Yaskawa INFORM job: SKRZYNIA_5440_180_STOPNI_10B_NEW.JBI

/JOB
//NAME SKRZYNIA_5440_180_STOPNI_10B_NEW
///FOLDERNAME 02-SKRZYNIE_JOBS
//POS
///NPOS 748,748,0,32,0,0
///TOOL 0
///POSTYPE PULSE
///PULSE
C00000=-21231,-51303,42314,2367,6591,-1439
C00001=-12854,-61498,-6635,149088,-29435,16513
C00002=84284,-61498,-6635,149088,14842,16513
C00003=84426,-61498,-62039,149088,14842,16513
C00004=84426,-61498,-83719,149088,14842,16513
C00005=40079,-25830,-61904,72398,37828,17494
C00006=40079,-25830,-61904,72398,37828,17494
C00007=38824,-23395,-60038,72349,38727,17731
C00008=41545,-22667,-59464,70826,37145,18191
C00009=40079,-25830,-61904,72398,37828,17494
C00010=40079,-23879,-31232,97616,36989,2612
C00011=40241,-22903,-30855,97033,36795,2952
C00012=39596,-21803,-29985,96678,37187,3182
C00013=41542,-21522,-29763,96797,35874,3054
C00014=40241,-22903,-30855,97033,36795,2952
C00015=44500,-22967,-34027,49689,40772,15208
C00016=44759,-21950,-33222,49364,40770,15399
C00017=43898,-20603,-32137,49608,41392,15289
C00018=45676,-20288,-31878,48567,40497,15854
C00019=44759,-21950,-33222,49364,40770,15399
C00020=50639,-31838,-53853,40430,42590,20636
C00021=47737,-42531,-47731,84740,46626,-3202
C00022=73324,-51450,-15857,136644,48513,-27329
C00023=28578,-31257,-33285,101874,54895,-3139
C00024=29101,-23166,-41439,93785,52323,3372
C00025=30342,-16402,-40775,90158,51109,6027
C00026=29555,-14242,-38855,90054,51607,6222
C00027=31304,-14182,-38798,89754,50458,6198
C00028=30342,-16402,-40775,90158,51109,6027
C00029=37840,-26567,-47806,97824,39338,5403
C00030=38314,-22656,-45541,96192,38787,6352
C00031=38740,-21749,-44817,95954,38481,6451
C00032=38106,-20505,-43805,95701,38856,6673
C00033=39920,-20274,-43616,95549,37666,6573
C00034=38740,-21749,-44817,95954,38481,6451
C00035=35154,-23288,-28184,89821,43405,2441
C00036=35403,-21021,-26397,89340,43215,2751
C00037=34678,-19569,-25213,89063,43699,2948
C00038=36545,-19419,-25091,89018,42427,2940
C00039=35403,-21021,-26397,89340,43215,2751
C00040=46673,-28267,-59493,36306,49500,22578
C00041=47298,-25083,-54483,36432,48421,22382
C00042=46134,-23276,-53085,36983,49197,22170
C00043=48093,-22778,-52692,35651,48513,22818
C00044=47298,-25083,-54483,36432,48421,22382
C00045=43000,-32780,-49011,53703,41088,15214
C00046=66148,-65994,-55487,105361,28212,-7739
C00047=66148,-65994,-55487,105361,28212,-7739
C00048=59848,-54778,-49507,133915,29212,-10807
C00049=45497,-38347,-41839,114412,32622,-465
C00050=46376,-32635,-46933,102993,29107,5780
C00051=46303,-28031,-46898,97061,28371,8976
C00052=45038,-26161,-45521,96183,29128,9541
C00053=46946,-25787,-45238,96120,27855,9431
C00054=46303,-28031,-46898,97061,28371,8976
C00055=45864,-17128,1685,129467,40696,-9274
C00056=46023,-15894,1830,128891,40053,-8896
C00057=45181,-14790,2774,128176,40341,-8535
C00058=46921,-14545,2986,129317,39465,-9073
C00059=45402,-17127,796,128656,40504,-8810
C00060=42828,-21985,-11573,106778,34538,-1929
C00061=43349,-21404,-11124,106831,34165,-1930
C00062=42250,-19876,-9917,105946,34757,-1485
C00063=44494,-19460,-9583,106781,33302,-1837
C00064=42797,-21858,-11474,106726,34550,-1903
C00065=42956,-14057,7354,88292,32197,-569
C00066=43438,-13569,7781,88275,31880,-510
C00067=42549,-12302,8904,87823,32462,-349
C00068=44721,-11883,9282,88161,31033,-316
C00069=42944,-14884,6642,88491,32210,-682
C00070=72417,-64226,-72669,53660,37323,27470
C00071=81480,-74508,-67932,111005,17511,3722
C00072=42492,-36415,-29790,92406,42740,11684
C00073=29699,-14901,-14062,86637,51249,15251
C00074=28921,-12904,-12269,86425,51786,15406
C00075=30978,-12767,-12144,86426,50380,15429
C00076=29506,-17416,-16239,86937,51377,15018
C00077=29506,-17416,-16239,86937,51377,15018
C00078=44296,-22319,-14791,77397,31382,16857
C00079=44081,-20100,-12685,77077,31564,17025
C00080=42936,-18463,-11353,76734,32387,17168
C00081=44621,-18276,-11197,76464,31271,17386
C00082=44081,-20100,-12685,77077,31564,17025
C00083=88410,-69609,-60867,139529,19008,-8209
C00084=82254,-59190,-37505,135829,26015,-2584
C00085=48709,-26647,-10027,118963,31871,904
C00086=44740,-24992,-19428,105622,30913,8023
C00087=35836,-10089,175,120717,54219,3716
C00088=33571,-11609,-5533,116057,52820,8482
C00089=32638,-9483,-3533,115639,53262,8773
C00090=34483,-9329,-3384,116184,52162,8425
C00091=33571,-11609,-5533,116057,52820,8482
C00092=29299,-14235,-8112,85858,51306,13749
C00093=30258,-13056,-7056,85778,50658,13854
C00094=29454,-11053,-5212,85557,51212,13988
C00095=31306,-10982,-5149,85624,49953,14016
C00096=30258,-13056,-7056,85778,50658,13854
C00097=44150,-27478,-14760,79983,38437,11062
C00098=60260,-41997,-20174,82745,25327,6782
C00099=62412,-62489,-12046,-12266,17816,34850
C00100=0,-52280,40443,0,6876,0
C00101=-681,-52632,38645,-5695,5489,-631
C00102=-17840,-61498,-6635,-149088,-29435,-16513
C00103=-84284,-61498,-6635,-149088,14842,-16513
C00104=-84426,-61498,-62039,-149088,14842,-16513
C00105=-84426,-61498,-83719,-149088,14842,-16513
C00106=-83351,-27062,-60322,-167360,37385,6517
C00107=-83351,-27062,-60322,-167360,37385,23281
C00108=-45097,-23850,-79932,-76262,26943,-22849
C00109=-48253,-15729,-73342,-71138,25693,-24842
C00110=-50302,-13076,-73239,-65836,25323,-27140
C00111=-49401,-11675,-71961,-66260,25816,-27133
C00112=-50608,-11574,-71867,-65226,25249,-27391
C00113=-49660,-13361,-73494,-66442,25615,-26975
C00114=-48242,-21102,-77802,-73044,25430,-23851
C00115=-42432,-29691,-46140,-101591,34194,-3953
C00116=-40467,-32259,-45349,-89481,35752,-6083
C00117=-35590,-22323,-38089,-87474,43148,-7978
C00118=-34853,-20780,-36847,-87247,43643,-8181
C00119=-37029,-20471,-36594,-86926,42180,-8224
C00120=-35503,-23333,-38886,-87700,43207,-7835
C00121=-41659,-25848,-37197,-61468,39541,-12344
C00122=-42019,-23363,-32043,-63110,38591,-11327
C00123=-41283,-22167,-31102,-63128,39154,-11341
C00124=-43189,-21868,-30866,-62281,38009,-11788
C00125=-40846,-25460,-35158,-62968,39555,-11455
C00126=-39561,-32409,-42051,-71473,38885,-9254
C00127=-88477,-67032,-53890,-125185,13082,17955
C00128=-90715,-66667,-50935,-152816,24533,28486
C00129=-30735,-26920,-32844,-95116,50209,-1071
C00130=-37180,-24683,-31930,-114741,47007,2943
C00131=-36407,-19634,-34656,-109847,45004,-453
C00132=-38352,-16604,-33863,-108521,43129,-1176
C00133=-37479,-14809,-32279,-108169,43576,-1482
C00134=-39395,-14487,-31992,-108361,42368,-1194
C00135=-37253,-18321,-35339,-108644,43916,-1187
C00136=-30948,-19486,-27368,-89515,49970,-2899
C00137=-32453,-17458,-25663,-89179,48933,-3088
C00138=-31896,-16151,-24534,-89028,49305,-3221
C00139=-33527,-16125,-24510,-88960,48196,-3202
C00140=-31291,-18911,-26892,-89421,49733,-2955
C00141=-32789,-14788,-10714,-75998,48642,-1904
C00142=-33953,-13481,-9550,-75758,47902,-2112
C00143=-33380,-12226,-8408,-75670,48319,-2157
C00144=-35020,-12164,-8351,-75529,47228,-2306
C00145=-33300,-14767,-10697,-75957,48300,-1949
C00146=-33300,-14767,-10697,-75957,48300,-1949
C00147=-33901,-13199,-7224,-76945,47663,-1266
C00148=-33178,-11617,-5779,-76815,48184,-1329
C00149=-35129,-11426,-5603,-76688,46886,-1497
C00150=-32900,-14718,-9841,-76444,48459,-1584
C00151=-46324,-38325,-53351,-48650,39022,-16558
C00152=-84678,-53272,-42524,-56273,5220,-14251
C00153=-79949,-57830,-54545,-43165,18800,-25262
C00154=-85199,-63426,-59279,-35356,8253,-25340
C00155=-43240,-40066,-69296,-76804,34492,-13950
C00156=-32352,-24302,-62495,-76398,48702,-17646
C00157=-33867,-19497,-59989,-74208,48202,-18898
C00158=-33043,-17469,-58279,-74274,48770,-19034
C00159=-35172,-17180,-58031,-73305,47532,-19251
C00160=-33150,-20833,-61090,-74721,48572,-18687
C00161=-32525,-19963,-22291,-97454,48417,-2656
C00162=-34479,-17146,-19937,-97221,47013,-2812
C00163=-33716,-15515,-18525,-96928,47480,-3025
C00164=-35357,-15455,-18472,-97073,46375,-2908
C00165=-33341,-18474,-21063,-97306,47817,-2759
C00166=-32838,-10388,7981,-94473,48357,2926
C00167=-33747,-9461,8037,-94117,47673,2571
C00168=-33094,-8062,9377,-93861,48090,2458
C00169=-34952,-7927,9507,-94260,46861,2543
C00170=-33010,-10379,7174,-94037,48174,2591
C00171=-36099,-20774,-22249,-70758,44565,-7624
C00172=-37926,-16067,-12890,-73276,42575,-5996
C00173=-37323,-14944,-11908,-73188,43017,-6038
C00174=-39053,-14785,-11769,-72915,41882,-6255
C00175=-37847,-19214,-17221,-72670,42783,-6386
C00176=-73757,-59015,-49060,-81128,17325,-3444
C00177=-66351,-49775,-22313,-134939,32824,19491
C00178=-38126,-18978,-6321,-103556,42156,4232
C00179=-39485,-17529,-8330,-90200,39091,223
C00180=-38315,-15563,-6658,-89669,39866,-39
C00181=-40130,-15376,-6497,-89855,38637,-21
C00182=-40610,-23081,-12745,-91737,38407,1092
C00183=-40833,-20771,-16117,-71062,38118,-5732
C00184=-41179,-17944,-14058,-70159,38104,-6286
C00185=-40208,-16344,-12701,-70049,38815,-6328
C00186=-42019,-16101,-12492,-69614,37653,-6637
C00187=-41179,-17944,-14058,-70159,38104,-6286
C00188=-82794,-45547,-18103,-153793,26453,27163
C00189=-59391,-59726,-723,-139936,47315,26256
C00190=-59391,-63256,-7305,-138930,45803,25558
C00191=-41911,-25348,-18707,-96909,37821,5942
C00192=-39278,-18921,-13723,-94727,39374,4724
C00193=-50267,-3803,20766,-145166,53580,20077
C00194=-49199,-2294,22340,-144514,53890,19722
C00195=-50839,-1881,22778,-145489,53339,20243
C00196=-50267,-457,30009,-146420,56926,21139
C00197=-39278,-18921,-13723,-94727,39374,4724
C00198=-38355,-17353,-12416,-94258,39960,4466
C00199=-40180,-17161,-12255,-94505,38724,4557
C00200=-37963,-22229,-16363,-95272,40353,5112
C00201=-56568,-73357,-35482,-123268,35826,13545
C00202=-46099,-67236,-11725,-98004,28606,19827
C00203=275,-40498,62911,330,272,-175
C00204=-21231,-51303,42314,2367,6591,-1439
C00205=-12854,-61498,-6635,149088,-29435,16513
C00206=84284,-61498,-6635,149088,14842,16513
C00207=84426,-61498,-62039,149088,14842,16513
C00208=84426,-61498,-83719,149088,14842,16513
C00209=40079,-25830,-61904,72398,37828,17494
C00210=43542,-21744,-53414,85694,32141,12908
C00211=43538,-20959,-59091,78847,32551,16732
C00212=40079,-23879,-31232,97616,36989,2612
C00213=41069,-22296,-36683,87871,35939,7163
C00214=41069,-20857,-27994,94343,36275,3375
C00215=40241,-22903,-30855,97033,36795,2952
C00216=44500,-22967,-34027,49689,40772,15208
C00217=37674,-14410,-29425,54908,51799,12689
C00218=37617,-13106,-20810,58248,49229,10178
C00219=44759,-21950,-33222,49364,40770,15399
C00220=50639,-31838,-53853,40430,42590,20636
C00221=47737,-42531,-47731,84740,46626,-3202
C00222=78713,-49095,-28754,133607,38203,-24422
C00223=28578,-31257,-33285,101874,54895,-3139
C00224=29101,-23166,-41439,93785,52323,3372
C00225=31163,-13872,-34138,92103,50752,4440
C00226=31163,-14064,-41434,88282,50498,7326
C00227=30342,-16402,-40775,90158,51109,6027
C00228=37840,-26567,-47806,97824,39338,5403
C00229=38314,-22656,-45541,96192,38787,6352
C00230=39658,-19881,-39017,99036,38353,4498
C00231=39658,-20227,-46296,93241,37598,7980
C00232=38740,-21749,-44817,95954,38481,6451
C00233=35154,-23288,-28184,89821,43405,2441
C00234=36302,-20456,-32356,81251,42995,6506
C00235=36302,-19046,-24537,85721,42698,3608
C00236=35403,-21021,-26397,89340,43215,2751
C00237=46673,-28267,-59493,36306,49500,22578
C00238=35383,-14910,-45807,52457,59655,19882
C00239=35383,-15025,-38926,54776,56903,17744
C00240=47298,-25083,-54483,36432,48421,22382
C00241=43000,-32780,-49011,53703,41088,15214
C00242=90538,-65158,-52413,145953,6697,-22013
C00243=90538,-65158,-52413,145953,6697,-22013
C00244=59848,-54778,-49507,133915,29212,-10807
C00245=45497,-38347,-41839,114412,32622,-465
C00246=46376,-32635,-46933,102993,29107,5780
C00247=38443,-20223,-37840,96971,39567,10287
C00248=38443,-20698,-44956,91660,38993,13539
C00249=46303,-28031,-46898,97061,28371,8976
C00250=45864,-17128,1685,129467,40696,-9274
C00251=38069,-7942,12691,120284,49952,-5070
C00252=38069,-11604,1369,116685,47266,-2469
C00253=45402,-17127,796,128656,40504,-8810
C00254=42828,-21985,-11573,106778,34538,-1929
C00255=33281,-15275,-13406,92642,47209,4970
C00256=33281,-12456,-2996,97026,47894,1870
C00257=42797,-21858,-11474,106726,34550,-1903
C00258=42956,-14057,7354,88292,32197,-569
C00259=35915,-8349,8335,81338,43542,2014
C00260=35915,-4149,20758,86814,43229,-1568
C00261=42944,-14884,6642,88491,32210,-682
C00262=72417,-64226,-72669,53660,37323,27470
C00263=81480,-74508,-67932,111005,17511,3722
C00264=42492,-36415,-29790,92406,42740,11684
C00265=30589,-12517,-11440,90322,50747,14596
C00266=30928,-12247,-10742,85035,50377,15419
C00267=29506,-17416,-16239,86937,51377,15018
C00268=33836,-18112,-25401,68178,50408,21159
C00269=33465,-13162,-18426,69063,50292,20506
C00270=33465,-11483,-10771,72168,49104,18208
C00271=88410,-69609,-60867,139529,19008,-8209
C00272=82254,-59190,-37505,135829,26015,-2584
C00273=48709,-26647,-10027,118963,31871,904
C00274=44740,-24992,-19428,105622,30913,8023
C00275=35836,-10089,175,120717,54219,3716
C00276=34345,-8030,793,117331,53206,7509
C00277=34322,-10419,-8163,114502,51063,9720
C00278=33571,-11609,-5533,116057,52820,8482
C00279=29299,-14235,-8112,85858,51306,13749
C00280=31207,-11656,-8788,84025,50108,15207
C00281=31207,-8775,1760,88103,49995,12167
C00282=30258,-13056,-7056,85778,50658,13854
C00283=44150,-27478,-14760,79983,38437,11062
C00284=60260,-41997,-20174,82745,25327,6782
C00285=62412,-62489,-12046,-12266,17816,34850
C00286=0,-52280,40443,0,6876,0
C00287=-681,-52632,38645,-5695,5489,-631
C00288=-17840,-61498,-6635,-149088,-29435,-16513
C00289=-84284,-61498,-6635,-149088,14842,-16513
C00290=-84426,-61498,-62039,-149088,14842,-16513
C00291=-84426,-61498,-83719,-149088,14842,-16513
C00292=-83351,-27062,-60322,-167360,37385,6517
C00293=-83351,-27062,-60322,-167360,37385,23281
C00294=-45097,-23850,-79932,-76262,26943,-22849
C00295=-48253,-15729,-73342,-71138,25693,-24842
C00296=-42869,-6204,-67496,-75794,33821,-25861
C00297=-42869,-3205,-70686,-69723,34977,-29338
C00298=-49660,-13361,-73494,-66442,25615,-26975
C00299=-48242,-21102,-77802,-73044,25430,-23851
C00300=-42432,-29691,-46140,-101591,34194,-3953
C00301=-40467,-32259,-45349,-89481,35752,-6083
C00302=-32032,-15700,-34761,-86363,49905,-9645
C00303=-32032,-14866,-27372,-89947,49973,-6979
C00304=-35503,-23333,-38886,-87700,43207,-7835
C00305=-41659,-25848,-37197,-61468,39541,-12344
C00306=-32550,-13183,-23016,-68651,53358,-8526
C00307=-34023,-12481,-22084,-63241,53452,-9524
C00308=-40846,-25460,-35158,-62968,39555,-11455
C00309=-39561,-32409,-42051,-71473,38885,-9254
C00310=-88477,-67032,-53890,-125185,13082,17955
C00311=-90715,-66667,-50935,-152816,24533,28486
C00312=-30735,-26920,-32844,-95116,50209,-1071
C00313=-37180,-24683,-31930,-114741,47007,2943
C00314=-36407,-19634,-34656,-109847,45004,-453
C00315=-39264,-14095,-28560,-110319,43249,69
C00316=-39254,-14742,-35710,-105973,41627,-2729
C00317=-37253,-18321,-35339,-108644,43916,-1187
C00318=-30948,-19486,-27368,-89515,49970,-2899
C00319=-33188,-17217,-33290,-80523,49125,-7157
C00320=-33231,-16133,-25752,-84153,48705,-4513
C00321=-31291,-18911,-26892,-89421,49733,-2955
C00322=-32789,-14788,-10714,-75998,48642,-1904
C00323=-32456,-10000,-8763,-74569,51725,-2878
C00324=-32456,-7502,814,-78111,50801,-165
C00325=-33300,-14767,-10697,-75957,48300,-1949
C00326=-33300,-14767,-10697,-75957,48300,-1949
C00327=-31039,-7597,-4415,-75714,54029,-1891
C00328=-31745,-5891,1281,-74609,53027,-1007
C00329=-32900,-14718,-9841,-76444,48459,-1584
C00330=-46324,-38325,-53351,-48650,39022,-16558
C00331=-84678,-53272,-42524,-56273,5220,-14251
C00332=-79949,-57830,-54545,-43165,18800,-25262
C00333=-85199,-63426,-59279,-35356,8253,-25340
C00334=-43240,-40066,-69296,-76804,34492,-13950
C00335=-32352,-24302,-62495,-76398,48702,-17646
C00336=-34311,-15084,-43386,-89458,46770,-12174
C00337=-34303,-14562,-49859,-85086,46777,-15220
C00338=-33150,-20833,-61090,-74721,48572,-18687
C00339=-32525,-19963,-22291,-97454,48417,-2656
C00340=-35706,-13608,-12356,-102024,46946,-662
C00341=-35706,-15621,-21438,-97808,45877,-3577
C00342=-33341,-18474,-21063,-97306,47817,-2759
C00343=-32838,-10388,7981,-94473,48357,2926
C00344=-33093,-7396,5806,-90907,49596,566
C00345=-33114,-3922,16616,-94789,50065,3444
C00346=-33010,-10379,7174,-94037,48174,2591
C00347=-36099,-20774,-22249,-70758,44565,-7624
C00348=-34715,-11750,-12273,-72011,49148,-6727
C00349=-34715,-9605,-3694,-75523,48112,-4187
C00350=-37847,-19214,-17221,-72670,42783,-6386
C00351=-73757,-59015,-49060,-81128,17325,-3444
C00352=-66351,-49775,-22313,-134939,32824,19491
C00353=-38126,-18978,-6321,-103556,42156,4232
C00354=-35411,-10902,-672,-92816,45935,848
C00355=-36000,-11295,-2683,-84848,44809,-1301
C00356=-40610,-23081,-12745,-91737,38407,1092
C00357=-46116,-25645,-29995,-54013,38610,-12898
C00358=-36364,-11468,-16502,-61524,50356,-10311
C00359=-36364,-9268,-6699,-65335,48232,-7516
C00360=-35369,-17970,-15673,-74843,50412,-3942
C00361=-82794,-45547,-18103,-153793,26453,27163
C00362=-59391,-59726,-723,-139936,47315,26256
///LIMIT ON
C00363=-59391,-69594,-18878,-137021,43274,24283
///LIMIT OFF
C00364=-41911,-25348,-18707,-96909,37821,5942
C00365=-39278,-18921,-13723,-94727,39374,4724
C00366=-41964,3488,28151,-134521,60914,14195
C00367=-41964,-819,15200,-132329,56719,12142
C00368=-50267,-457,30009,-146420,56926,21139
C00369=-33715,-10212,-1364,-94538,48612,5206
C00370=-33715,-12585,-10220,-90890,48191,2581
C00371=-37963,-22229,-16363,-95272,40353,5112
C00372=-66368,-73811,-34662,-141094,38161,28545
C00373=-46099,-67236,-11725,-98004,28606,19827
C00374=275,-40498,62911,330,272,-175
C00375=-21231,-51303,42314,2367,6591,-1439
C00376=-12854,-61498,-6635,149088,-29435,16513
C00377=32880,-72586,-50560,79734,53940,25582
C00378=76664,-93599,-96338,114349,24908,7990
C00379=72545,-76403,-90681,98079,12187,16258
C00380=68435,-42241,-79282,43384,21203,43145
C00381=65057,-16377,-54230,51764,24572,24912
C00382=65057,-16377,-54230,51764,24572,24912
C00383=63338,-14509,-52578,53100,25585,24479
C00384=65493,-13068,-51269,50530,24633,25485
C00385=65057,-16377,-54230,51764,24572,24912
C00386=65057,-15356,-24189,99795,20011,765
C00387=64877,-14372,-23690,98704,20045,1316
C00388=64002,-13489,-22890,98156,20604,1621
C00389=65592,-12702,-22173,98357,19527,1466
C00390=64877,-14372,-23690,98704,20045,1316
C00391=68341,-13254,-25781,29903,31229,25524
C00392=68283,-12212,-24821,29865,31356,25548
C00393=67188,-11145,-23825,30867,31841,25051
C00394=68624,-10377,-23095,29361,31405,25809
C00395=68283,-12212,-24821,29865,31356,25548
C00396=67373,-28813,-51747,26561,36937,27500
C00397=65665,-56911,-59086,75825,31170,1181
C00398=86238,-56758,-47218,93606,16664,-7096
C00399=86238,-56758,-47218,93606,16664,-7096
C00400=58162,-25487,-29222,106212,35121,-6052
C00401=54729,-17550,-36821,90686,35172,3055
C00402=53879,-10723,-35593,84994,35691,6442
C00403=52628,-8898,-33837,85063,36512,6546
C00404=54193,-8333,-33282,84633,35489,6620
C00405=53879,-10723,-35593,84994,35691,6442
C00406=63265,-18185,-41125,95483,22448,4389
C00407=62561,-14368,-38517,92984,22773,5727
C00408=62689,-13396,-37636,92694,22678,5861
C00409=61812,-12400,-36718,92465,23238,6064
C00410=63331,-11679,-36046,92201,22238,6052
C00411=62689,-13396,-37636,92694,22678,5861
C00412=60836,-16142,-22303,87853,25853,3109
C00413=60346,-13901,-20318,87240,26185,3441
C00414=59279,-12702,-19226,86999,26911,3593
C00415=60868,-12050,-18626,86765,25831,3679
C00416=60346,-13901,-20318,87240,26185,3441
C00417=71174,-16943,-50501,16787,44328,31924
C00418=70846,-13961,-45205,17496,43056,31510
C00419=69412,-12602,-43961,18675,43507,30969
C00420=70949,-11616,-43043,17320,43301,31610
C00421=70846,-13961,-45205,17496,43056,31510
C00422=66765,-25643,-43957,33958,30926,25005
C00423=89904,-51519,-74342,14421,36812,44678
C00424=59533,-60921,-66479,83565,41795,11392
C00425=74572,-27669,-34920,136415,14797,-11887
C00426=72479,-21736,-38943,108586,11547,1590
C00427=70901,-17325,-38411,94105,11830,8638
C00428=69318,-15905,-37172,92885,12849,9347
C00429=70820,-15051,-36412,92531,11846,9399
C00430=70901,-17325,-38411,94105,11830,8638
C00431=70927,-7523,10343,151197,29871,-19432
C00432=70517,-6236,10737,150221,29352,-18933
C00433=69462,-5331,11645,148944,29606,-18324
C00434=70849,-4645,12343,150548,29173,-19084
C00435=70402,-7634,9356,150158,29478,-18907
C00436=68660,-13051,-4106,122816,18275,-8999
C00437=68895,-12351,-3471,122899,18094,-9031
C00438=67458,-11121,-2337,120787,18802,-8043
C00439=69212,-10147,-1425,122703,17774,-8922
C00440=68590,-12934,-4000,122687,18305,-8939
C00441=67960,-5141,15741,92957,15720,-628
C00442=68207,-4523,16370,92944,15555,-601
C00443=67051,-3465,17460,92338,16311,-404
C00444=68762,-2475,18496,92897,15183,-531
C00445=68227,-5981,14898,93242,15553,-745
C00446=75423,-38775,-29488,68062,11357,11878
C00447=83800,-53438,-37305,103753,14733,-1265
C00448=73693,-37430,-30368,101200,21937,8332
C00449=54083,-9583,-9164,86048,34613,15862
C00450=52816,-7862,-7494,85864,35484,15962
C00451=54627,-7152,-6792,85763,34247,16030
C00452=54668,-12069,-11504,86415,34208,15656
C00453=56304,-11796,-18615,61131,36292,25169
C00454=55378,-9761,-17250,60867,37124,25353
C00455=54231,-8210,-15746,61227,37881,25175
C00456=56022,-7436,-14984,60355,36824,25634
C00457=55378,-9761,-17250,60867,37124,25353
C00458=89016,-59505,-36896,143842,20811,-11822
C00459=60495,-76741,-47652,120298,37447,-3273
C00460=76037,-16315,-2108,148598,17507,-12246
C00461=70560,-15452,-11753,122116,14270,428
C00462=55952,-2531,9844,130476,44298,-1945
C00463=56211,-3395,4409,126223,41962,1193
C00464=55729,-3443,2508,124592,39934,3479
C00465=57337,-2775,3210,125461,39069,2998
C00466=55715,-2364,6430,126525,43399,286
C00467=54062,-9026,-3291,86300,34474,14396
C00468=54568,-7612,-1915,86151,34132,14497
C00469=53276,-5879,-187,85948,35014,14576
C00470=54919,-5291,406,85945,33897,14626
C00471=54568,-7612,-1915,86151,34132,14497
C00472=55516,-30048,-16468,81245,30784,11190
C00473=78642,-41617,-20006,83725,13431,8209
C00474=0,-52280,40443,0,6876,0
C00475=-681,-52632,38645,-5695,5489,-631
C00476=-17840,-61498,-6635,-149088,-29435,-16513
C00477=-84284,-61498,-6635,-149088,14842,-16513
C00478=-57949,-92832,-68327,-119114,39180,-13331
C00479=-51160,-78996,-68705,-103851,38676,-21739
C00480=-70129,-12201,-70194,-45988,15849,-32683
C00481=-70861,-4247,-62448,-43170,16032,-33903
C00482=-72229,-1292,-61598,-37253,16795,-36501
C00483=-71164,-286,-60510,-39045,17142,-35862
C00484=-72168,114,-60071,-37345,16819,-36474
C00485=-71747,-1710,-62044,-38091,16943,-36199
C00486=-72086,-8949,-67137,-41785,15362,-34318
C00487=-68226,-19972,-38714,-103620,16923,-1218
C00488=-67549,-22986,-38612,-80975,17520,-9124
C00489=-60286,-14955,-31870,-81576,26630,-9634
C00490=-59206,-13694,-30736,-81541,27366,-9725
C00491=-61026,-12796,-29913,-80837,26167,-9971
C00492=-60502,-15936,-32740,-81790,26471,-9505
C00493=-66711,-16726,-29834,-42060,26790,-21996
C00494=-66477,-14329,-24475,-44917,25565,-20507
C00495=-65503,-13376,-23611,-45716,26132,-20127
C00496=-67048,-12587,-22889,-44009,25442,-20959
C00497=-66009,-16611,-27996,-44380,26285,-20808
C00498=-67084,-23473,-35621,-52822,22843,-18344
C00499=-54372,-63877,-56403,-90862,27079,1323
C00500=-55608,-75012,-34654,-126966,55573,20814
C00501=-55608,-75012,-34654,-126966,55573,20814
C00502=-58069,-20780,-28125,-95622,31565,-134
C00503=-62818,-16895,-25617,-123146,31403,8811
C00504=-60301,-12189,-28106,-114654,29999,4030
C00505=-61167,-8731,-26593,-112607,28768,2985
C00506=-59960,-7252,-25135,-111997,29446,2563
C00507=-61574,-6413,-24296,-112502,28453,2957
C00508=-60636,-10677,-28466,-112685,29164,2987
C00509=-55814,-13636,-22293,-87541,33030,-3263
C00510=-56566,-11270,-20110,-87077,32519,-3496
C00511=-55709,-10167,-19066,-86969,33101,-3589
C00512=-57154,-9687,-18605,-86794,32120,-3632
C00513=-55949,-12989,-21706,-87412,32939,-3330
C00514=-57109,-8613,-4995,-71756,32687,-5152
C00515=-57764,-7017,-3429,-71410,32292,-5358
C00516=-56909,-5946,-2356,-71529,32873,-5273
C00517=-58347,-5433,-1836,-71115,31941,-5534
C00518=-57555,-8453,-4841,-71622,32398,-5235
C00519=-57555,-8453,-4841,-71622,32398,-5235
C00520=-57844,-6749,-1100,-73475,31868,-4209
C00521=-56760,-5394,262,-73573,32605,-4123
C00522=-58439,-4668,1002,-73167,31507,-4396
C00523=-57269,-8513,-4090,-72514,32435,-4729
C00524=-74194,-26905,-45748,-21164,30431,-30370
C00525=-93036,-61583,-83098,-4972,39040,-38907
C00526=-93036,-61583,-83098,-4972,39040,-38907
C00527=-71878,-28414,-61729,-48672,19032,-25171
C00528=-58025,-17185,-56692,-61796,34178,-22014
C00529=-58138,-12270,-53641,-59720,34855,-23185
C00530=-56898,-10637,-52111,-60384,35596,-23031
C00531=-58712,-9745,-51261,-58987,34681,-23500
C00532=-57851,-13714,-54968,-60141,34926,-22995
C00533=-57767,-13689,-16896,-100181,31334,-836
C00534=-58645,-10437,-13885,-99794,30663,-1040
C00535=-57513,-9065,-12573,-99347,31388,-1300
C00536=-58947,-8556,-12078,-99591,30423,-1148
C00537=-58031,-12031,-15383,-99926,31110,-974
C00538=-57646,-4162,14084,-101426,32077,4804
C00539=-58050,-2999,14481,-100683,31666,4357
C00540=-57067,-1784,15765,-100255,32298,4198
C00541=-58672,-1130,16464,-100866,31256,4407
C00542=-57676,-4116,13320,-100600,31921,4338
C00543=-61201,-13510,-16039,-60848,29053,-13371
C00544=-61885,-8475,-5914,-65722,27292,-10768
C00545=-61040,-7537,-4993,-65975,27855,-10622
C00546=-62506,-6917,-4380,-65230,26947,-11038
C00547=-62587,-11561,-10517,-63923,27184,-11731
C00548=-69972,-70945,-58827,-87515,19733,-17
C00549=-69972,-70945,-58827,-87515,19733,-17
C00550=-64053,-11295,342,-114563,25508,8776
C00551=-64305,-9514,-1154,-92513,22236,350
C00552=-62690,-7882,422,-91839,23314,70
C00553=-64201,-7220,1072,-92034,22288,112
C00554=-67149,-14673,-5883,-94845,20391,1413
C00555=-66316,-14019,-26011,-36889,31466,-23117
C00556=-65553,-11798,-21321,-39176,30584,-21892
C00557=-64393,-10599,-20193,-40085,31193,-21437
C00558=-66059,-9659,-19295,-38481,30526,-22253
C00559=-65553,-11798,-21321,-39176,30584,-21892
C00560=-66017,-67071,-29713,-134523,32873,22112
C00561=-66017,-67071,-29713,-134523,48860,22112
C00562=-66017,-67071,-29713,-134523,48860,22112
C00563=-68464,-16512,-11702,-102583,19802,8050
C00564=-64069,-10918,-6685,-98748,22529,6223
C00565=-71808,7543,33524,-159735,48317,27747
C00566=-70546,8877,35161,-158835,48660,27285
C00567=-71854,9797,36309,-159820,48523,27800
C00568=-71808,11433,44144,-160620,52560,28413
C00569=-64069,-10918,-6685,-98748,22529,6223
C00570=-62794,-9626,-5461,-98007,23355,5872
C00571=-64311,-8958,-4821,-98397,22329,6039
C00572=-64031,-14482,-9933,-99750,22651,6736
C00573=-78219,-66180,-35295,-149347,29259,30999
C00574=-46099,-67236,-11725,-98004,28606,19827
C00575=275,-40498,62911,330,272,-175
C00576=-21231,-51303,42314,2367,6591,-1439
C00577=-12854,-61498,-6635,149088,-29435,16513
C00578=84284,-61498,-6635,149088,14842,16513
C00579=84426,-61498,-62039,149088,14842,16513
C00580=84426,-61498,-83719,149088,14842,16513
C00581=65057,-16377,-54230,51764,24572,24912
C00582=84197,-12836,-45810,-45141,8815,68584
C00583=84197,-12041,-51210,-30828,12194,61758
C00584=65057,-15356,-24189,99795,20011,765
C00585=74080,-15423,-30907,69143,7686,14038
C00586=74080,-14352,-23480,100923,7503,-991
C00587=64877,-14372,-23690,98704,20045,1316
C00588=68341,-13254,-25781,29903,31229,25524
C00589=74439,-11496,-26749,13621,29642,33649
C00590=74439,-10401,-19085,15788,25340,32499
C00591=68283,-12212,-24821,29865,31356,25548
C00592=75452,-19560,-44582,17787,36745,31835
C00593=68183,-44834,-62310,40554,34116,19994
C00594=94103,-63119,-69903,16230,17694,31762
C00595=91219,-55958,-51219,93435,14423,-1742
C00596=58162,-25487,-29222,106212,35121,-6052
C00597=54729,-17550,-36821,90686,35172,3055
C00598=70769,-15160,-35297,83470,11760,4000
C00599=70769,-15377,-40609,67973,12489,11436
C00600=53879,-10723,-35593,84994,35691,6442
C00601=63265,-18185,-41125,95483,22448,4389
C00602=62561,-14368,-38517,92984,22773,5727
C00603=77715,-13962,-33882,144680,4496,-21400
C00604=77806,-14046,-41277,60589,2532,18064
C00605=62689,-13396,-37636,92694,22678,5861
C00606=60836,-16142,-22303,87853,25853,3109
C00607=74678,-16514,-29029,42946,9451,23276
C00608=74678,-15315,-21920,65026,7151,12815
C00609=60346,-13901,-20318,87240,26185,3441
C00610=71174,-16943,-50501,16787,44328,31924
C00611=80494,-13102,-44599,-1731,38384,44653
C00612=80494,-13295,-38861,-1907,34285,44756
C00613=70846,-13961,-45205,17496,43056,31510
C00614=69645,-22678,-41665,30358,30421,26767
C00615=81017,-78801,-66317,80675,7786,2447
C00616=81017,-78801,-66317,80675,7786,2447
C00617=74572,-27669,-34920,136415,14797,-11887
C00618=72479,-21736,-38943,108586,11547,1590
C00619=76162,-15538,-34076,119407,5153,-4143
C00620=76225,-15803,-40874,66675,4586,20654
C00621=70901,-17325,-38411,94105,11830,8638
C00622=70927,-7523,10343,151197,29871,-19432
C00623=75273,-951,23395,164730,33684,-27271
C00624=75257,-4812,11918,163197,28775,-26429
C00625=70402,-7634,9356,150158,29478,-18907
C00626=68660,-13051,-4106,122816,18275,-8999
C00627=75422,-13779,-12311,124767,7049,-10125
C00628=75402,-11409,-3274,143452,10422,-18986
C00629=68590,-12934,-4000,122687,18305,-8939
C00630=67960,-5141,15741,92957,15720,-628
C00631=77005,-5383,11265,73049,3770,10304
C00632=77005,-1367,23224,135174,5603,-18901
C00633=68227,-5981,14898,93242,15553,-745
C00634=83595,-66668,-34414,154325,14846,-28455
C00635=83595,-66668,-34414,154325,14846,-28455
C00636=69137,-30288,-25983,94330,24536,11676
C00637=73329,-13700,-12516,109108,8203,5807
C00638=73329,-11353,-3574,130600,10679,-4409
C00639=74337,-14270,-6219,134594,10484,-6281
C00640=76918,-16529,-25927,11673,20080,42529
C00641=75405,-13221,-23238,13992,20934,41419
C00642=75405,-11863,-15892,17135,17051,39858
C00643=46050,-47732,-32699,100114,41423,7030
C00644=72866,-68602,-36981,132032,32409,-7906
C00645=72866,-68602,-36981,132032,32409,-7906
C00646=76037,-16315,-2108,148598,17507,-12246
C00647=70560,-15452,-11753,122116,14270,428
C00648=58783,-935,13382,132999,43851,-3406
C00649=72693,-1568,14493,161814,36543,-14367
C00650=75650,3978,23428,169507,44505,-15919
C00651=70596,-8585,4037,153028,29768,-12051
C00652=54062,-9026,-3291,86300,34474,14396
C00653=70728,-11880,-8994,79432,11308,18593
C00654=70728,-9344,357,101276,11563,8141
C00655=54568,-7612,-1915,86151,34132,14497
C00656=62643,-28068,-15160,80125,26114,12294
C00657=92151,-29067,-13111,41177,6909,29587
C00658=79691,-50270,-13176,-792,17881,39424
C00659=0,-52280,40443,0,6876,0
C00660=-681,-52632,38645,-5695,5489,-631
C00661=-17840,-61498,-6635,-149088,-29435,-16513
C00662=-84284,-61498,-6635,-149088,14842,-16513
C00663=-84426,-61498,-62039,-149088,14842,-16513
C00664=-84426,-61498,-83719,-149088,14842,-16513
C00665=-83351,-27062,-60322,-167360,37385,6517
C00666=-83351,-27062,-60322,-167360,37385,23281
C00667=-70129,-12201,-70194,-45988,15849,-32683
C00668=-70861,-4247,-62448,-43170,16032,-33903
C00669=-76882,43,-60950,-14294,14755,-45201
C00670=-76882,3984,-64926,-10429,20329,-47102
C00671=-71747,-1710,-62044,-38091,16943,-36199
C00672=-72086,-8949,-67137,-41785,15362,-34318
C00673=-68226,-19972,-38714,-103620,16923,-1218
C00674=-67549,-22986,-38612,-80975,17520,-9124
C00675=-69143,-15166,-34287,-68804,15212,-14794
C00676=-69143,-14592,-28782,-80821,14459,-8960
C00677=-60502,-15936,-32740,-81790,26471,-9505
C00678=-66711,-16726,-29834,-42060,26790,-21996
C00679=-75652,-13136,-22972,-17539,18443,-33643
C00680=-76393,-11602,-18975,-13556,19574,-34543
C00681=-66009,-16611,-27996,-44380,26285,-20808
C00682=-61601,-28306,-39228,-59626,25389,-15050
C00683=-72315,-63222,-70224,-69600,33305,-10426
C00684=-72315,-63222,-70224,-69600,33305,-10426
C00685=-58069,-20780,-28125,-95622,31565,-134
C00686=-62818,-16895,-25617,-123146,31403,8811
C00687=-60301,-12189,-28106,-114654,29999,4030
C00688=-75089,-9933,-24682,-148597,14783,22922
C00689=-75089,-10642,-34451,-132584,9653,15243
C00690=-60636,-10677,-28466,-112685,29164,2987
C00691=-55814,-13636,-22293,-87541,33030,-3263
C00692=-73301,-16058,-32281,-44459,12702,-22095
C00693=-73339,-15052,-25249,-60236,10249,-14543
C00694=-55949,-12989,-21706,-87412,32939,-3330
C00695=-57109,-8613,-4995,-71756,32687,-5152
C00696=-71674,-10355,-9102,-48278,15013,-17468
C00697=-71670,-8088,-356,-62615,12652,-10541
C00698=-57555,-8453,-4841,-71622,32398,-5235
C00699=-57555,-8453,-4841,-71622,32398,-5235
C00700=-73349,-10209,-7254,-46090,12597,-18565
C00701=-73349,-7867,1452,-63091,10217,-10432
C00702=-57269,-8513,-4090,-72514,32435,-4729
C00703=-74194,-26905,-45748,-21164,30431,-30370
C00704=-76007,-77202,-67157,-59280,11041,-11579
C00705=-76006,-77203,-67157,-59281,11043,-11581
C00706=-53398,-42726,-55849,-45492,34374,-18069
C00707=-71878,-28414,-61729,-48672,19032,-25171
C00708=-58025,-17185,-56692,-61796,34178,-22014
C00709=-77553,-14661,-43008,-35465,5780,-31120
C00710=-77553,-14004,-50514,-17997,10868,-39389
C00711=-57851,-13714,-54968,-60141,34926,-22995
C00712=-57767,-13689,-16896,-100181,31334,-836
C00713=-74769,-11126,-10073,-142523,13426,19686
C00714=-74753,-12848,-17783,-130765,10301,14051
C00715=-58031,-12031,-15383,-99926,31110,-974
C00716=-57646,-4162,14084,-101426,32077,4804
C00717=-72179,-7124,6017,-115427,12582,9833
C00718=-72179,-4103,15503,-129018,15105,16401
C00719=-57676,-4116,13320,-100600,31921,4338
C00720=-61201,-13510,-16039,-60848,29053,-13371
C00721=-74136,-10643,-11909,-32993,14820,-27251
C00722=-74162,-8377,-2780,-45377,11297,-21290
C00723=-62587,-11561,-10517,-63923,27184,-11731
C00724=-68334,-63389,-52515,-83837,20864,-1739
C00725=-68334,-63389,-52515,-83837,20864,-1739
C00726=-64053,-11295,342,-114563,25508,8776
C00727=-75758,-9453,-2048,-123101,7379,13416
C00728=-76003,-8378,955,-106758,5948,6887
C00729=-77335,-11553,-2051,-113345,5246,9938
C00730=-79087,-12138,-19852,-4327,22551,-37435
C00731=-78014,-10681,-18487,-6037,22777,-36592
C00732=-78014,-8816,-9327,-7606,17906,-35805
C00733=-78501,-19622,-30273,-4965,24122,-37125
C00734=-65551,-48104,-28924,-114827,24376,11665
C00735=-39771,-60653,-24362,-111239,58263,14171
C00736=-39771,-60652,-24363,-111239,58260,14167
C00737=-68464,-16512,-11702,-102583,19802,8050
C00738=-64069,-10918,-6685,-98748,22529,6223
C00739=-75794,5019,20382,-166088,42002,32193
C00740=-75794,5019,20382,-166088,42002,32193
C00741=-71808,11433,44144,-160620,52560,28413
C00742=-74529,-9237,-439,-131085,10959,21329
C00743=-74560,-11298,-8213,-120962,9324,16064
C00744=-64031,-14482,-9933,-99750,22651,6736
C00745=-65667,-47452,-26760,-125785,27682,20101
C00746=-46099,-67236,-11725,-98004,28606,19827
C00747=275,-40498,62911,330,272,-175
BC00000=467225
BC00001=513669
BC00002=494109
BC00003=467540
BC00004=467540
BC00005=478876
BC00006=478876
BC00007=478876
BC00008=478876
BC00009=478876
BC00010=478876
BC00011=478876
BC00012=478876
BC00013=478876
BC00014=478876
BC00015=478876
BC00016=478876
BC00017=478876
BC00018=478876
BC00019=478876
BC00020=478876
BC00021=481980
BC00022=563952
BC00023=606256
BC00024=606256
BC00025=606252
BC00026=606252
BC00027=606252
BC00028=606252
BC00029=654662
BC00030=654618
BC00031=654618
BC00032=654618
BC00033=654618
BC00034=654618
BC00035=654618
BC00036=654618
BC00037=654618
BC00038=654618
BC00039=654618
BC00040=686402
BC00041=686402
BC00042=686350
BC00043=686350
BC00044=686402
BC00045=652574
BC00046=648164
BC00047=761837
BC00048=784046
BC00049=784046
BC00050=784046
BC00051=784046
BC00052=784046
BC00053=784046
BC00054=784046
BC00055=784046
BC00056=784046
BC00057=784046
BC00058=784046
BC00059=784046
BC00060=821134
BC00061=821134
BC00062=821134
BC00063=821134
BC00064=821134
BC00065=821134
BC00066=821134
BC00067=821134
BC00068=821134
BC00069=821134
BC00070=849627
BC00071=945583
BC00072=909600
BC00073=909600
BC00074=909600
BC00075=909600
BC00076=909600
BC00077=924128
BC00078=924128
BC00079=924128
BC00080=924128
BC00081=924128
BC00082=924128
BC00083=945583
BC00084=1035849
BC00085=1030374
BC00086=1030374
BC00087=1021815
BC00088=1021652
BC00089=1021652
BC00090=1021652
BC00091=1021652
BC00092=1021652
BC00093=1021652
BC00094=1021652
BC00095=1021652
BC00096=1021652
BC00097=1012294
BC00098=1002860
BC00099=923175
BC00100=828403
BC00101=518986
BC00102=509920
BC00103=467540
BC00104=467540
BC00105=467540
BC00106=521167
BC00107=520352
BC00108=535759
BC00109=535759
BC00110=535757
BC00111=535757
BC00112=535757
BC00113=535757
BC00114=535757
BC00115=485653
BC00116=485653
BC00117=485653
BC00118=485653
BC00119=485653
BC00120=485653
BC00121=485653
BC00122=485653
BC00123=485653
BC00124=485653
BC00125=485653
BC00126=485653
BC00127=485653
BC00128=615112
BC00129=615112
BC00130=615112
BC00131=615112
BC00132=615112
BC00133=615112
BC00134=615112
BC00135=615112
BC00136=615112
BC00137=615112
BC00138=615112
BC00139=615112
BC00140=615112
BC00141=615112
BC00142=615112
BC00143=615112
BC00144=615112
BC00145=615112
BC00146=658076
BC00147=658076
BC00148=658076
BC00149=658076
BC00150=658076
BC00151=655680
BC00152=643721
BC00153=643721
BC00154=793396
BC00155=799070
BC00156=799070
BC00157=799070
BC00158=799070
BC00159=799070
BC00160=799070
BC00161=799070
BC00162=799070
BC00163=799070
BC00164=799070
BC00165=799070
BC00166=799070
BC00167=799070
BC00168=799070
BC00169=799070
BC00170=799070
BC00171=845667
BC00172=845667
BC00173=845667
BC00174=845667
BC00175=845667
BC00176=845667
BC00177=899436
BC00178=899436
BC00179=899436
BC00180=899436
BC00181=899436
BC00182=899436
BC00183=924302
BC00184=924302
BC00185=924302
BC00186=924302
BC00187=924302
BC00188=899436
BC00189=862979
BC00190=1007989
BC00191=1038788
BC00192=1038788
BC00193=1025790
BC00194=1025790
BC00195=1025790
BC00196=1025790
BC00197=1038788
BC00198=1038788
BC00199=1038788
BC00200=1038788
BC00201=1022413
BC00202=926201
BC00203=639407
BC00204=467225
BC00205=513669
BC00206=494109
BC00207=467540
BC00208=467540
BC00209=478876
BC00210=478876
BC00211=478876
BC00212=478876
BC00213=478876
BC00214=478876
BC00215=478876
BC00216=478876
BC00217=478876
BC00218=478876
BC00219=478876
BC00220=478876
BC00221=481980
BC00222=594876
BC00223=606256
BC00224=606256
BC00225=606252
BC00226=606252
BC00227=606252
BC00228=654662
BC00229=654618
BC00230=654618
BC00231=654618
BC00232=654618
BC00233=654618
BC00234=654618
BC00235=654618
BC00236=654618
BC00237=686402
BC00238=686402
BC00239=686402
BC00240=686402
BC00241=652574
BC00242=641414
BC00243=715810
BC00244=784046
BC00245=784046
BC00246=784046
BC00247=784046
BC00248=784046
BC00249=784046
BC00250=784046
BC00251=784043
BC00252=784043
BC00253=784046
BC00254=821134
BC00255=821134
BC00256=821134
BC00257=821134
BC00258=821134
BC00259=821134
BC00260=821134
BC00261=821134
BC00262=849627
BC00263=945583
BC00264=909600
BC00265=909600
BC00266=909600
BC00267=913824
BC00268=932344
BC00269=932344
BC00270=932344
BC00271=945583
BC00272=1035849
BC00273=1030374
BC00274=1030374
BC00275=1021815
BC00276=1021652
BC00277=1021652
BC00278=1021652
BC00279=1021652
BC00280=1021652
BC00281=1021652
BC00282=1021652
BC00283=1012294
BC00284=1002860
BC00285=923175
BC00286=828403
BC00287=518986
BC00288=509920
BC00289=467540
BC00290=467540
BC00291=467540
BC00292=521167
BC00293=520352
BC00294=535759
BC00295=535759
BC00296=535757
BC00297=535757
BC00298=535757
BC00299=535757
BC00300=485653
BC00301=485653
BC00302=485653
BC00303=485653
BC00304=485653
BC00305=485653
BC00306=485653
BC00307=485653
BC00308=485653
BC00309=485653
BC00310=485653
BC00311=615112
BC00312=615112
BC00313=615112
BC00314=615112
BC00315=615112
BC00316=615112
BC00317=615112
BC00318=615112
BC00319=615112
BC00320=615112
BC00321=615112
BC00322=615112
BC00323=615112
BC00324=615112
BC00325=615112
BC00326=658076
BC00327=658076
BC00328=658076
BC00329=658076
BC00330=655680
BC00331=643721
BC00332=643721
BC00333=793396
BC00334=799070
BC00335=799070
BC00336=799070
BC00337=799070
BC00338=799070
BC00339=799070
BC00340=799070
BC00341=799070
BC00342=799070
BC00343=799070
BC00344=799070
BC00345=799070
BC00346=799070
BC00347=845667
BC00348=845667
BC00349=845667
BC00350=845667
BC00351=845667
BC00352=899436
BC00353=899436
BC00354=899436
BC00355=899436
BC00356=899436
BC00357=922093
BC00358=922093
BC00359=922093
BC00360=919368
BC00361=899436
BC00362=862979
BC00363=1007989
BC00364=1038788
BC00365=1038788
BC00366=1025790
BC00367=1025790
BC00368=1025790
BC00369=1038788
BC00370=1038788
BC00371=1038788
BC00372=1038788
BC00373=895479
BC00374=639407
BC00375=467225
BC00376=513669
BC00377=542621
BC00378=535309
BC00379=478364
BC00380=478364
BC00381=478876
BC00382=478876
BC00383=478876
BC00384=478876
BC00385=478876
BC00386=478876
BC00387=478876
BC00388=478876
BC00389=478876
BC00390=478876
BC00391=478876
BC00392=478876
BC00393=478876
BC00394=478876
BC00395=478876
BC00396=478876
BC00397=480759
BC00398=480759
BC00399=560395
BC00400=606256
BC00401=606256
BC00402=606252
BC00403=606252
BC00404=606252
BC00405=606252
BC00406=654662
BC00407=654618
BC00408=654618
BC00409=654618
BC00410=654618
BC00411=654618
BC00412=654618
BC00413=654618
BC00414=654618
BC00415=654618
BC00416=654618
BC00417=686402
BC00418=686402
BC00419=686350
BC00420=686350
BC00421=686402
BC00422=652574
BC00423=652574
BC00424=774850
BC00425=784046
BC00426=784046
BC00427=784046
BC00428=784046
BC00429=784046
BC00430=784046
BC00431=784046
BC00432=784046
BC00433=784046
BC00434=784046
BC00435=784046
BC00436=821134
BC00437=821134
BC00438=821134
BC00439=821134
BC00440=821134
BC00441=821134
BC00442=821134
BC00443=821134
BC00444=821134
BC00445=821134
BC00446=821134
BC00447=846623
BC00448=909600
BC00449=909600
BC00450=909600
BC00451=909600
BC00452=909600
BC00453=934865
BC00454=934865
BC00455=934865
BC00456=934865
BC00457=934865
BC00458=909600
BC00459=1025782
BC00460=1030374
BC00461=1030374
BC00462=1021815
BC00463=1021652
BC00464=1021652
BC00465=1021652
BC00466=1021652
BC00467=1021652
BC00468=1021652
BC00469=1021652
BC00470=1021652
BC00471=1021652
BC00472=1012294
BC00473=1002860
BC00474=859125
BC00475=518986
BC00476=509920
BC00477=467540
BC00478=497868
BC00479=497868
BC00480=535759
BC00481=535759
BC00482=535757
BC00483=535757
BC00484=535757
BC00485=535757
BC00486=535757
BC00487=485653
BC00488=485653
BC00489=485653
BC00490=485653
BC00491=485653
BC00492=485653
BC00493=485653
BC00494=485653
BC00495=485653
BC00496=485653
BC00497=485653
BC00498=485653
BC00499=485653
BC00500=485653
BC00501=601945
BC00502=615112
BC00503=615112
BC00504=615112
BC00505=615112
BC00506=615112
BC00507=615112
BC00508=615112
BC00509=615112
BC00510=615112
BC00511=615112
BC00512=615112
BC00513=615112
BC00514=615112
BC00515=615112
BC00516=615112
BC00517=615112
BC00518=615112
BC00519=658076
BC00520=658076
BC00521=658076
BC00522=658076
BC00523=658076
BC00524=655680
BC00525=655680
BC00526=765678
BC00527=799070
BC00528=799070
BC00529=799070
BC00530=799070
BC00531=799070
BC00532=799070
BC00533=799070
BC00534=799070
BC00535=799070
BC00536=799070
BC00537=799070
BC00538=799070
BC00539=799070
BC00540=799070
BC00541=799070
BC00542=799070
BC00543=845667
BC00544=845667
BC00545=845667
BC00546=845667
BC00547=845667
BC00548=845667
BC00549=900547
BC00550=899436
BC00551=899436
BC00552=899436
BC00553=899436
BC00554=899436
BC00555=930438
BC00556=930438
BC00557=930438
BC00558=930438
BC00559=930438
BC00560=899436
BC00561=943124
BC00562=1002282
BC00563=1038788
BC00564=1038788
BC00565=1025790
BC00566=1025790
BC00567=1025790
BC00568=1025790
BC00569=1038788
BC00570=1038788
BC00571=1038788
BC00572=1038788
BC00573=1038788
BC00574=926201
BC00575=639407
BC00576=467225
BC00577=513669
BC00578=494109
BC00579=467540
BC00580=467540
BC00581=478876
BC00582=478876
BC00583=478876
BC00584=478876
BC00585=478876
BC00586=478876
BC00587=478876
BC00588=478876
BC00589=478876
BC00590=478876
BC00591=478876
BC00592=478876
BC00593=479530
BC00594=502776
BC00595=571156
BC00596=606256
BC00597=606256
BC00598=606252
BC00599=606252
BC00600=606252
BC00601=654662
BC00602=654618
BC00603=654618
BC00604=654618
BC00605=654618
BC00606=654618
BC00607=654618
BC00608=654618
BC00609=654618
BC00610=686402
BC00611=686402
BC00612=686402
BC00613=686402
BC00614=652574
BC00615=654591
BC00616=763025
BC00617=784046
BC00618=784046
BC00619=784046
BC00620=784046
BC00621=784046
BC00622=784046
BC00623=784043
BC00624=784043
BC00625=784046
BC00626=821134
BC00627=821134
BC00628=821134
BC00629=821134
BC00630=821134
BC00631=821134
BC00632=821134
BC00633=821134
BC00634=821134
BC00635=884766
BC00636=909600
BC00637=909600
BC00638=909600
BC00639=909600
BC00640=935274
BC00641=935274
BC00642=935274
BC00643=909600
BC00644=909600
BC00645=1002742
BC00646=1030374
BC00647=1030374
BC00648=1021815
BC00649=1021652
BC00650=1021652
BC00651=1021652
BC00652=1021652
BC00653=1021652
BC00654=1021652
BC00655=1021652
BC00656=1012294
BC00657=1002860
BC00658=951590
BC00659=828403
BC00660=518986
BC00661=509920
BC00662=467540
BC00663=467540
BC00664=467540
BC00665=521167
BC00666=520352
BC00667=535759
BC00668=535759
BC00669=535757
BC00670=535757
BC00671=535757
BC00672=535757
BC00673=485653
BC00674=485653
BC00675=485653
BC00676=485653
BC00677=485653
BC00678=485653
BC00679=485653
BC00680=485653
BC00681=485653
BC00682=485653
BC00683=485653
BC00684=600333
BC00685=615112
BC00686=615112
BC00687=615112
BC00688=615112
BC00689=615112
BC00690=615112
BC00691=615112
BC00692=615112
BC00693=615112
BC00694=615112
BC00695=615112
BC00696=615112
BC00697=615112
BC00698=615112
BC00699=658076
BC00700=658076
BC00701=658076
BC00702=658076
BC00703=655680
BC00704=656245
BC00705=762546
BC00706=762546
BC00707=799070
BC00708=799070
BC00709=799070
BC00710=799070
BC00711=799070
BC00712=799070
BC00713=799070
BC00714=799070
BC00715=799070
BC00716=799070
BC00717=799070
BC00718=799070
BC00719=799070
BC00720=845667
BC00721=845667
BC00722=845667
BC00723=845667
BC00724=845667
BC00725=902133
BC00726=899436
BC00727=899436
BC00728=899436
BC00729=899436
BC00730=928010
BC00731=928010
BC00732=928010
BC00733=928010
BC00734=899436
BC00735=899436
BC00736=1012029
BC00737=1038788
BC00738=1038788
BC00739=1039249
BC00740=1031057
BC00741=1025790
BC00742=1038788
BC00743=1038788
BC00744=1038788
BC00745=1038788
BC00746=926201
BC00747=639407
///POSTYPE BASE
///RECTAN
///RCONF 1,0,0,0,0,0,0,0,0,0,0,0,0,0,0,0,0,0,0,0,0,0,0,0
P00006=0.000,0.000,0.000,0.0000,0.0000,0.0000
///RCONF 0,0,0,0,0,0,0,0,0,0,0,0,0,0,0,0,0,0,0,0,0,0,0,0
P00056=0.000,0.000,5.000,0.0000,0.0000,0.0000
///RCONF 1,0,0,0,0,0,0,0,0,0,0,0,0,0,0,0,0,0,0,0,0,0,0,0
P00301=0.046,-2.112,7.779,0.0000,0.0000,0.0000
P00302=-0.180,-2.409,6.326,0.0000,0.0000,0.0000
///RCONF 0,0,0,0,0,0,0,0,0,0,0,0,0,0,0,0,0,0,0,0,0,0,0,0
P00303=-0.004,-1.437,-4.584,0.0000,0.0000,0.0000
P00304=0.028,-1.666,-4.234,0.0000,0.0000,0.0000
P00305=-0.003,-1.920,-3.501,0.0000,0.0000,0.0000
P00306=0.015,-2.252,-3.054,0.0000,0.0000,0.0000
P00307=0.019,-2.151,-5.077,0.0000,0.0000,0.0000
P00308=-0.003,-2.092,-4.888,0.0000,0.0000,0.0000
P00309=-0.040,-2.205,-4.992,0.0000,0.0000,0.0000
P00310=-0.006,-2.490,-5.925,0.0000,0.0000,0.0000
P00311=-0.007,-2.079,-5.307,0.0000,0.0000,0.0000
P00312=-0.032,2.202,-7.632,0.0000,0.0000,0.0000
///RCONF 1,0,0,0,0,0,0,0,0,0,0,0,0,0,0,0,0,0,0,0,0,0,0,0
P00313=-0.088,1.055,2.110,0.0000,0.0000,0.0000
P00314=-0.055,1.752,1.634,0.0000,0.0000,0.0000
P00318=-0.086,2.132,2.037,0.0000,0.0000,0.0000
///RCONF 0,0,0,0,0,0,0,0,0,0,0,0,0,0,0,0,0,0,0,0,0,0,0,0
P00351=13.563,-0.027,-0.653,0.0000,0.0000,0.0000
P00352=13.252,-0.027,-0.827,0.0000,0.0000,0.0000
P00353=10.971,-0.082,0.776,0.0000,0.0000,0.0000
P00354=-0.024,2.508,-1.824,0.0000,0.0000,0.0000
P00355=-0.001,2.528,-1.131,0.0000,0.0000,0.0000
P00356=-0.034,2.921,-0.262,0.0000,0.0000,0.0000
P00357=0.003,3.386,-0.091,0.0000,0.0000,0.0000
P00358=0.014,3.037,-0.020,0.0000,0.0000,0.0000
P00359=-0.005,2.731,0.912,0.0000,0.0000,0.0000
P00360=-0.011,3.412,0.438,0.0000,0.0000,0.0000
P00361=0.018,3.050,1.253,0.0000,0.0000,0.0000
P00362=0.014,2.784,0.148,0.0000,0.0000,0.0000
P00363=0.026,4.310,-2.639,0.0000,0.0000,0.0000
P00364=0.034,4.181,-4.040,0.0000,0.0000,0.0000
P00380=-0.012,-4.857,1.526,0.0000,0.0000,0.0000
//INST
///DATE 2024/05/21 11:34
///ATTR SC,RW
///GROUP1 RB1,BS1
NOP
CALL JOB:MOVE_INTO_TUNNEL
MOVJ C00000 BC00000 VJ=10.00
MOVJ C00001 BC00001 VJ=10.00
MOVJ C00002 BC00002 VJ=10.00
MOVJ C00003 BC00003 VJ=10.00
MOVJ C00004 BC00004 VJ=10.00
'------------------------
'W29.2
'------------------------
MOVL C00005 BC00005 V=500.0
'------------------------
'W63.5
'------------------------
SFTOF
MOVL C00006 BC00006 V=166.7 PL=0
REFP 3 C00007 BC00007
CALL JOB:SEARCH-R1
IMOV P0056 V=50.0 PL=0
SET P0301 P0006
SFTON P0301
REFP 3 C00008 BC00008
CALL JOB:SEARCH-R1
SET P0301 P0006
SFTON P0301
MOVL C00009 BC00009 V=166.7 PL=0
SFTOF
MOVL C00010 BC00010 V=500.0
MOVL C00011 BC00011 V=166.7 PL=0
REFP 3 C00012 BC00012
CALL JOB:SEARCH-R1
IMOV P0056 V=50.0 PL=0
SET P0302 P0006
SFTON P0302
REFP 3 C00013 BC00013
CALL JOB:SEARCH-R1
SET P0302 P0006
SFTON P0302
MOVL C00014 BC00014 V=166.7 PL=0
SFTOF
MOVL C00015 BC00015 V=500.0
MOVL C00016 BC00016 V=166.7 PL=0
REFP 3 C00017 BC00017
CALL JOB:SEARCH-R1
IMOV P0056 V=50.0 PL=0
SET P0303 P0006
SFTON P0303
REFP 3 C00018 BC00018
CALL JOB:SEARCH-R1
SET P0303 P0006
SFTON P0303
SFTOF
MOVL C00019 BC00019 V=166.7 PL=0
MOVL C00020 BC00020 V=500.0
MOVJ C00021 BC00021 VJ=30.00
MOVJ C00022 BC00022 VJ=30.00
MOVJ C00023 BC00023 VJ=30.00
MOVL C00024 BC00024 V=500.0
'------------------------
'W29.14
'------------------------
MOVL C00025 BC00025 V=166.7 PL=0
REFP 3 C00026 BC00026
CALL JOB:SEARCH-R1
IMOV P0056 V=23.0 PL=0
SET P0304 P0006
SFTON P0304
REFP 3 C00027 BC00027
CALL JOB:SEARCH-R1
SET P0304 P0006
SFTON P0304
MOVL C00028 BC00028 V=66.7 PL=0
SFTOF
'PRZEJAZD
MOVL C00029 BC00029 V=500.0
MOVL C00030 BC00030 V=500.0
'------------------------
'W63.17
'------------------------
MOVL C00031 BC00031 V=166.7 PL=0
REFP 3 C00032 BC00032
CALL JOB:SEARCH-R1
IMOV P0056 V=23.0 PL=0
SET P0305 P0006
SFTON P0305
REFP 3 C00033 BC00033
CALL JOB:SEARCH-R1
SET P0305 P0006
SFTON P0305
MOVL C00034 BC00034 V=166.7 PL=0
SFTOF
MOVL C00035 BC00035 V=500.0
MOVL C00036 BC00036 V=166.7
REFP 3 C00037 BC00037
CALL JOB:SEARCH-R1
IMOV P0056 V=23.0 PL=0
SET P0306 P0006
SFTON P0306
REFP 3 C00038 BC00038
CALL JOB:SEARCH-R1
SET P0306 P0006
SFTON P0306
MOVL C00039 BC00039 V=166.7 PL=0
'PRZEJAZD
MOVL C00040 BC00040 V=500.0
MOVL C00041 BC00041 V=166.7
REFP 3 C00042 BC00042
CALL JOB:SEARCH-R1
IMOV P0056 V=23.0 PL=0
SET P0307 P0006
SFTON P0307
REFP 3 C00043 BC00043
CALL JOB:SEARCH-R1
SET P0307 P0006
SFTON P0307
MOVL C00044 BC00044 V=166.7 PL=0
SFTOF
MOVJ C00045 BC00045 VJ=20.00
MOVJ C00046 BC00046 VJ=20.00
MOVJ C00047 BC00047 VJ=30.00
MOVJ C00048 BC00048 VJ=30.00
MOVJ C00049 BC00049 VJ=30.00
MOVL C00050 BC00050 V=500.0
'------------------------
'W63.20
'------------------------
MOVL C00051 BC00051 V=166.7 PL=0
REFP 3 C00052 BC00052
CALL JOB:SEARCH-R1
IMOV P0056 V=23.0 PL=0
SET P0308 P0006
SFTON P0308
REFP 3 C00053 BC00053
CALL JOB:SEARCH-R1
SET P0308 P0006
SFTON P0308
MOVL C00054 BC00054 V=166.7 PL=0
SFTOF
'PRZEJAZD
MOVL C00055 BC00055 V=500.0
'------------------------
'W63.23
'------------------------
MOVL C00056 BC00056 V=166.7 PL=0
REFP 3 C00057 BC00057
CALL JOB:SEARCH-R1
IMOV P0056 V=23.0 PL=0
SET P0309 P0006
SFTON P0309
REFP 3 C00058 BC00058
CALL JOB:SEARCH-R1
SET P0309 P0006
SFTON P0309
MOVL C00059 BC00059 V=250.0 PL=0
SFTOF
MOVL C00060 BC00060 V=500.0
MOVL C00061 BC00061 V=166.7 PL=0
REFP 3 C00062 BC00062
CALL JOB:SEARCH-R1
IMOV P0056 V=23.0 PL=0
SET P0310 P0006
SFTON P0310
REFP 3 C00063 BC00063
CALL JOB:SEARCH-R1
SET P0310 P0006
SFTON P0310
MOVL C00064 BC00064 V=250.0 PL=0
SFTOF
MOVL C00065 BC00065 V=500.0
MOVL C00066 BC00066 V=166.7 PL=0
REFP 3 C00067 BC00067
CALL JOB:SEARCH-R1
IMOV P0056 V=23.0 PL=0
SET P0311 P0006
SFTON P0311
REFP 3 C00068 BC00068
CALL JOB:SEARCH-R1
SET P0311 P0006
SFTON P0311
MOVL C00069 BC00069 V=250.0 PL=0
SFTOF
MOVL C00070 BC00070 V=500.0
MOVL C00071 BC00071 V=500.0
MOVL C00072 BC00072 V=333.3
'------------------------
'W29.29
'------------------------
MOVL C00073 BC00073 V=166.7 PL=0
REFP 3 C00074 BC00074
CALL JOB:SEARCH-R1
IMOV P0056 V=23.0 PL=0
SET P0312 P0006
SFTON P0312
REFP 3 C00075 BC00075
CALL JOB:SEARCH-R1
SET P0312 P0006
SFTON P0312
MOVL C00076 BC00076 V=250.0 PL=0
SFTOF
MOVL C00077 BC00077 V=333.3
MOVL C00078 BC00078 V=333.3
MOVL C00079 BC00079 V=166.7
REFP 3 C00080 BC00080
CALL JOB:SEARCH-R1
IMOV P0056 V=23.0 PL=0
SET P0318 P0006
SFTON P0318
REFP 3 C00081 BC00081
CALL JOB:SEARCH-R1
SET P0318 P0006
SFTON P0318
MOVL C00082 BC00082 V=250.0 PL=0
SFTOF
'PRZEJAZD
MOVL C00083 BC00083 V=333.3
'PRZEJAZD
MOVL C00084 BC00084 V=500.0
MOVL C00085 BC00085 V=500.0
MOVL C00086 BC00086 V=333.3
MOVL C00087 BC00087 V=333.3
MOVL C00088 BC00088 V=166.7 PL=0
REFP 3 C00089 BC00089
CALL JOB:SEARCH-R1
IMOV P0056 V=23.0 PL=0
SET P0313 P0006
SFTON P0313
REFP 3 C00090 BC00090
CALL JOB:SEARCH-R1
SET P0313 P0006
SFTON P0313
MOVL C00091 BC00091 V=250.0 PL=0
SFTOF
MOVL C00092 BC00092 V=333.3
MOVL C00093 BC00093 V=166.7 PL=0
REFP 3 C00094 BC00094
CALL JOB:SEARCH-R1
IMOV P0056 V=23.0 PL=0
SET P0314 P0006
SFTON P0314
REFP 3 C00095 BC00095
CALL JOB:SEARCH-R1
SET P0314 P0006
SFTON P0314
MOVL C00096 BC00096 V=250.0 PL=0
SFTOF
MOVJ C00097 BC00097 VJ=10.00
MOVJ C00098 BC00098 VJ=10.00
MOVJ C00099 BC00099 VJ=30.00
MOVJ C00100 BC00100 VJ=20.00
MOVJ C00101 BC00101 VJ=50.00
MOVJ C00102 BC00102 VJ=20.00
MOVJ C00103 BC00103 VJ=10.00
MOVJ C00104 BC00104 VJ=20.00
MOVJ C00105 BC00105 VJ=20.00
'------------------------
'W28.2
'------------------------
MOVJ C00106 BC00106 VJ=10.00
MOVJ C00107 BC00107 VJ=10.00
MOVL C00108 BC00108 V=500.0
MOVL C00109 BC00109 V=500.0
'------------------------
'W62.5
'------------------------
MOVL C00110 BC00110 V=166.7 PL=0
REFP 3 C00111 BC00111
CALL JOB:SEARCH-R1
IMOV P0056 V=23.0 PL=0
SET P0351 P0006
SFTON P0351
REFP 3 C00112 BC00112
CALL JOB:SEARCH-R1
SET P0351 P0006
SFTON P0351
MOVL C00113 BC00113 V=250.0 PL=0
SFTOF
'PRZEJAZD
MOVL C00114 BC00114 V=500.0
MOVL C00115 BC00115 V=500.0
MOVL C00116 BC00116 V=500.0
MOVL C00117 BC00117 V=166.7 PL=0
REFP 3 C00118 BC00118
CALL JOB:SEARCH-R1
IMOV P0056 V=23.0 PL=0
SET P0352 P0006
SFTON P0352
REFP 3 C00119 BC00119
CALL JOB:SEARCH-R1
SET P0352 P0006
SFTON P0352
MOVL C00120 BC00120 V=250.0 PL=0
SFTOF
MOVL C00121 BC00121 V=500.0
'------------------------
'W29.8
'------------------------
MOVL C00122 BC00122 V=166.7 PL=0
REFP 3 C00123 BC00123
CALL JOB:SEARCH-R1
IMOV P0056 V=23.0 PL=0
SET P0353 P0006
SFTON P0353
REFP 3 C00124 BC00124
CALL JOB:SEARCH-R1
SET P0353 P0006
SFTON P0353
MOVL C00125 BC00125 V=250.0 PL=0
SFTOF
MOVL C00126 BC00126 V=500.0
'PRZEJAZD
MOVL C00127 BC00127 V=500.0
MOVJ C00128 BC00128 VJ=20.00
MOVL C00129 BC00129 V=500.0
MOVL C00130 BC00130 V=500.0
MOVL C00131 BC00131 V=500.0
'------------------------
'W29.11
'------------------------
MOVL C00132 BC00132 V=166.7 PL=0
REFP 3 C00133 BC00133
CALL JOB:SEARCH-R1
IMOV P0056 V=23.0 PL=0
SET P0354 P0006
SFTON P0354
REFP 3 C00134 BC00134
CALL JOB:SEARCH-R1
SET P0354 P0006
SFTON P0354
MOVL C00135 BC00135 V=250.0 PL=0
SFTOF
'PRZEJAZD
MOVL C00136 BC00136 V=500.0
'------------------------
'W29.14
'------------------------
MOVL C00137 BC00137 V=166.7 PL=0
REFP 3 C00138 BC00138
CALL JOB:SEARCH-R1
IMOV P0056 V=23.0 PL=0
SET P0355 P0006
SFTON P0355
REFP 3 C00139 BC00139
CALL JOB:SEARCH-R1
SET P0355 P0006
SFTON P0355
MOVL C00140 BC00140 V=250.0 PL=0
SFTOF
'PRZEJAZD
MOVL C00141 BC00141 V=500.0
'------------------------
'W63.17
'------------------------
MOVL C00142 BC00142 V=166.7 PL=0
REFP 3 C00143 BC00143
CALL JOB:SEARCH-R1
IMOV P0056 V=23.0 PL=0
SET P0356 P0006
SFTON P0356
REFP 3 C00144 BC00144
CALL JOB:SEARCH-R1
SET P0356 P0006
SFTON P0356
MOVL C00145 BC00145 V=250.0 PL=0
SFTOF
MOVL C00146 BC00146 V=500.0
MOVL C00147 BC00147 V=166.7 PL=0
REFP 3 C00148 BC00148
CALL JOB:SEARCH-R1
IMOV P0056 V=23.0 PL=0
SET P0357 P0006
SFTON P0357
REFP 3 C00149 BC00149
CALL JOB:SEARCH-R1
SET P0357 P0006
SFTON P0357
MOVL C00150 BC00150 V=250.0 PL=0
SFTOF
'PRZEJAZD
MOVL C00151 BC00151 V=500.0
MOVJ C00152 BC00152 VJ=30.00
MOVJ C00153 BC00153 VJ=30.00
MOVJ C00154 BC00154 VJ=30.00
MOVL C00155 BC00155 V=500.0
MOVL C00156 BC00156 V=500.0
'------------------------
'W62.20
'------------------------
MOVL C00157 BC00157 V=166.7 PL=0
REFP 3 C00158 BC00158
CALL JOB:SEARCH-R1
IMOV P0056 V=23.0 PL=0
SET P0358 P0006
SFTON P0358
REFP 3 C00159 BC00159
CALL JOB:SEARCH-R1
SET P0358 P0006
SFTON P0358
MOVL C00160 BC00160 V=250.0 PL=0
SFTOF
'PRZEJAZD
MOVL C00161 BC00161 V=500.0
'------------------------
'W63.23
'------------------------
MOVL C00162 BC00162 V=166.7 PL=0
REFP 3 C00163 BC00163
CALL JOB:SEARCH-R1
IMOV P0056 V=23.0 PL=0
SET P0359 P0006
SFTON P0359
REFP 3 C00164 BC00164
CALL JOB:SEARCH-R1
SET P0359 P0006
SFTON P0359
MOVL C00165 BC00165 V=250.0 PL=0
MOVL C00166 BC00166 V=500.0
'------------------------
'W29.29
'------------------------
MOVL C00167 BC00167 V=166.7 PL=0
REFP 3 C00168 BC00168
CALL JOB:SEARCH-R1
IMOV P0056 V=23.0 PL=0
SET P0360 P0006
SFTON P0360
REFP 3 C00169 BC00169
CALL JOB:SEARCH-R1
SET P0360 P0006
SFTON P0360
MOVL C00170 BC00170 V=250.0 PL=0
SFTOF
'PRZEJAZD
MOVL C00171 BC00171 V=500.0
MOVL C00172 BC00172 V=166.7 PL=0
REFP 3 C00173 BC00173
CALL JOB:SEARCH-R1
IMOV P0056 V=23.0 PL=0
SET P0361 P0006
SFTON P0361
REFP 3 C00174 BC00174
CALL JOB:SEARCH-R1
SET P0361 P0006
SFTON P0361
MOVL C00175 BC00175 V=250.0 PL=0
SFTOF
'------------------------
'W29.32
'------------------------
'PRZEJAZD
MOVL C00176 BC00176 V=500.0
MOVJ C00177 BC00177 VJ=10.00
MOVL C00178 BC00178 V=416.7
MOVL C00179 BC00179 V=166.7 PL=0
REFP 3 C00180 BC00180
CALL JOB:SEARCH-R1
IMOV P0056 V=23.0 PL=0
SET P0362 P0006
SFTON P0362
REFP 3 C00181 BC00181
CALL JOB:SEARCH-R1
SET P0362 P0006
SFTON P0362
MOVL C00182 BC00182 V=250.0 PL=0
SFTOF
MOVL C00183 BC00183 V=333.3
MOVL C00184 BC00184 V=166.7 PL=0
REFP 3 C00185 BC00185
CALL JOB:SEARCH-R1
IMOV P0056 V=23.0 PL=0
SET P0380 P0006
SFTON P0380
REFP 3 C00186 BC00186
CALL JOB:SEARCH-R1
SET P0380 P0006
SFTON P0380
MOVL C00187 BC00187 V=250.0 PL=0
SFTOF
MOVJ C00188 BC00188 VJ=20.00
MOVJ C00189 BC00189 VJ=30.00
MOVJ C00190 BC00190 VJ=30.00
MOVJ C00191 BC00191 VJ=15.00
MOVL C00192 BC00192 V=333.3
MOVL C00193 BC00193 V=250.0 PL=0
REFP 3 C00194 BC00194
CALL JOB:SEARCH-R1
IMOV P0056 V=23.0 PL=0
SET P0363 P0006
SFTON P0363
REFP 3 C00195 BC00195
CALL JOB:SEARCH-R1
SET P0363 P0006
SFTON P0363
MOVL C00196 BC00196 V=250.0 PL=0
SFTOF
MOVL C00197 BC00197 V=166.7 PL=0
REFP 3 C00198 BC00198
CALL JOB:SEARCH-R1
IMOV P0056 V=23.0 PL=0
SET P0364 P0006
SFTON P0364
REFP 3 C00199 BC00199
CALL JOB:SEARCH-R1
SET P0364 P0006
SFTON P0364
MOVL C00200 BC00200 V=250.0 PL=0
SFTOF
MOVJ C00201 BC00201 VJ=20.00
MOVJ C00202 BC00202 VJ=30.00
MOVJ C00203 BC00203 VJ=30.00
'KONIEC SEARCH WEW STRONA
MOVJ C00204 BC00204 VJ=30.00
MOVJ C00205 BC00205 VJ=20.00
MOVJ C00206 BC00206 VJ=10.00
MOVJ C00207 BC00207 VJ=20.00
MOVJ C00208 BC00208 VJ=20.00
'------------------------
'W29.2
'------------------------
MOVL C00209 BC00209 V=500.0
'------------------------
'W63.5
MACRO1 MJ#(0) ARGF9
'------------------------
SFTOF
SFTON P0301
MOVL C00210 BC00210 V=166.7 PL=0
ARCON
MOVL C00211 BC00211 V=10.0
ARCOF
SFTOF
MOVL C00212 BC00212 V=500.0
SFTON P0302
MOVL C00213 BC00213 V=166.7 PL=0
ARCON
MOVL C00214 BC00214 V=10.0
ARCOF
MOVL C00215 BC00215 V=166.7 PL=0
SFTOF
MOVL C00216 BC00216 V=500.0
SFTON P0303
MOVL C00217 BC00217 V=166.7 PL=0
ARCON
MOVL C00218 BC00218 V=10.0
ARCOF
SFTOF
MOVL C00219 BC00219 V=166.7 PL=0
MOVL C00220 BC00220 V=500.0
MOVJ C00221 BC00221 VJ=30.00
MOVJ C00222 BC00222 VJ=30.00
MOVJ C00223 BC00223 VJ=30.00
MOVL C00224 BC00224 V=500.0
'------------------------
'W29.14
'------------------------
SFTON P0304
MOVL C00225 BC00225 V=166.7 PL=0
ARCON
MOVL C00226 BC00226 V=10.0
ARCOF
MOVL C00227 BC00227 V=166.7 PL=0
SFTOF
'PRZEJAZD
MOVL C00228 BC00228 V=500.0
MOVL C00229 BC00229 V=500.0
'------------------------
'W63.17
'------------------------
SFTON P0305
MOVL C00230 BC00230 V=166.7 PL=0
ARCON
MOVL C00231 BC00231 V=10.0
ARCOF
MOVL C00232 BC00232 V=166.7 PL=0
SFTOF
MOVL C00233 BC00233 V=500.0
SFTON P0306
MOVL C00234 BC00234 V=166.7
ARCON
MOVL C00235 BC00235 V=10.0
ARCOF
MOVL C00236 BC00236 V=166.7 PL=0
SFTOF
'PRZEJAZD
MOVL C00237 BC00237 V=500.0
SFTON P0307
MOVL C00238 BC00238 V=166.7
ARCON
MOVL C00239 BC00239 V=10.0
ARCOF
MOVL C00240 BC00240 V=166.7 PL=0
SFTOF
MOVJ C00241 BC00241 VJ=20.00
MOVJ C00242 BC00242 VJ=20.00
MOVJ C00243 BC00243 VJ=30.00
MOVJ C00244 BC00244 VJ=30.00
MOVJ C00245 BC00245 VJ=30.00
MOVL C00246 BC00246 V=500.0
'------------------------
'W63.20
'------------------------
SFTON P0308
MOVL C00247 BC00247 V=166.7 PL=0
ARCON
MOVL C00248 BC00248 V=10.0
ARCOF
MOVL C00249 BC00249 V=166.7 PL=0
SFTOF
'PRZEJAZD
MOVL C00250 BC00250 V=500.0
'------------------------
'W63.23
'------------------------
SFTON P0309
MOVL C00251 BC00251 V=166.7 PL=0
ARCON
MOVL C00252 BC00252 V=10.0
ARCOF
MOVL C00253 BC00253 V=250.0 PL=0
SFTOF
MOVL C00254 BC00254 V=500.0
SFTON P0310
MOVL C00255 BC00255 V=166.7 PL=0
ARCON
MOVL C00256 BC00256 V=10.0
ARCOF
MOVL C00257 BC00257 V=250.0 PL=0
SFTOF
MOVL C00258 BC00258 V=500.0
SFTON P0311
MOVL C00259 BC00259 V=166.7 PL=0
ARCON
MOVL C00260 BC00260 V=10.0
ARCOF
MOVL C00261 BC00261 V=250.0 PL=0
SFTOF
MOVL C00262 BC00262 V=500.0
MOVL C00263 BC00263 V=500.0
MOVL C00264 BC00264 V=333.3
'------------------------
'W29.29
'------------------------
SFTON P0312
MOVL C00265 BC00265 V=166.7 PL=0
ARCON
MOVL C00266 BC00266 V=10.0
ARCOF
MOVL C00267 BC00267 V=250.0 PL=0
SFTOF
MOVL C00268 BC00268 V=250.0
SFTON P0318
MOVL C00269 BC00269 V=250.0
ARCON
MOVL C00270 BC00270 V=10.0
ARCOF
SFTOF
'PRZEJAZD
MOVL C00271 BC00271 V=333.3
'PRZEJAZD
'KONIEC SPAWANIA CZESCI WSPOLNEJ
MOVL C00272 BC00272 V=500.0
MOVL C00273 BC00273 V=500.0
MOVL C00274 BC00274 V=333.3
MOVL C00275 BC00275 V=333.3
SFTON P0313
MOVL C00276 BC00276 V=166.7 PL=0
ARCON
MOVL C00277 BC00277 V=10.0
ARCOF
MOVL C00278 BC00278 V=250.0 PL=0
SFTOF
MOVL C00279 BC00279 V=333.3
SFTON P0314
MOVL C00280 BC00280 V=166.7 PL=0
ARCON
MOVL C00281 BC00281 V=10.0
ARCOF
MOVL C00282 BC00282 V=250.0 PL=0
SFTOF
MOVJ C00283 BC00283 VJ=10.00
MOVJ C00284 BC00284 VJ=10.00
MOVJ C00285 BC00285 VJ=30.00
MOVJ C00286 BC00286 VJ=20.00
MOVJ C00287 BC00287 VJ=50.00
MOVJ C00288 BC00288 VJ=20.00
MOVJ C00289 BC00289 VJ=10.00
MOVJ C00290 BC00290 VJ=20.00
MOVJ C00291 BC00291 VJ=20.00
'------------------------
'W28.2
'------------------------
MOVJ C00292 BC00292 VJ=10.00
MOVJ C00293 BC00293 VJ=10.00
MOVL C00294 BC00294 V=500.0
MOVL C00295 BC00295 V=500.0
'------------------------
'W62.5
'------------------------
SFTON P0351
MOVL C00296 BC00296 V=166.7 PL=0
ARCON
MOVL C00297 BC00297 V=10.0
ARCOF
MOVL C00298 BC00298 V=250.0 PL=0
SFTOF
'PRZEJAZD
MOVL C00299 BC00299 V=500.0
MOVL C00300 BC00300 V=500.0
MOVL C00301 BC00301 V=500.0
SFTON P0352
MOVL C00302 BC00302 V=166.7 PL=0
ARCON
MOVL C00303 BC00303 V=10.0
ARCOF
MOVL C00304 BC00304 V=250.0 PL=0
SFTOF
MOVL C00305 BC00305 V=500.0
'------------------------
'W29.8
'------------------------
SFTON P0353
MOVL C00306 BC00306 V=166.7 PL=0
ARCON
MOVL C00307 BC00307 V=10.0
ARCOF
MOVL C00308 BC00308 V=250.0 PL=0
SFTOF
MOVL C00309 BC00309 V=500.0
'PRZEJAZD
MOVL C00310 BC00310 V=500.0
MOVJ C00311 BC00311 VJ=20.00
MOVL C00312 BC00312 V=500.0
MOVL C00313 BC00313 V=500.0
MOVL C00314 BC00314 V=500.0
'------------------------
'W29.11
'------------------------
SFTON P0354
MOVL C00315 BC00315 V=166.7 PL=0
ARCON
MOVL C00316 BC00316 V=10.0
ARCOF
MOVL C00317 BC00317 V=250.0 PL=0
SFTOF
'PRZEJAZD
MOVL C00318 BC00318 V=500.0
'------------------------
'W29.14
'------------------------
SFTON P0355
MOVL C00319 BC00319 V=166.7 PL=0
ARCON
MOVL C00320 BC00320 V=10.0
ARCOF
MOVL C00321 BC00321 V=250.0 PL=0
SFTOF
'PRZEJAZD
MOVL C00322 BC00322 V=500.0
'------------------------
'W63.17
'------------------------
SFTON P0356
MOVL C00323 BC00323 V=166.7 PL=0
ARCON
MOVL C00324 BC00324 V=10.0
ARCOF
MOVL C00325 BC00325 V=250.0 PL=0
SFTOF
MOVL C00326 BC00326 V=500.0
SFTON P0357
MOVL C00327 BC00327 V=166.7 PL=0
ARCON
MOVL C00328 BC00328 V=10.0
ARCOF
MOVL C00329 BC00329 V=250.0 PL=0
SFTOF
'PRZEJAZD
MOVL C00330 BC00330 V=500.0
MOVJ C00331 BC00331 VJ=30.00
MOVJ C00332 BC00332 VJ=30.00
MOVJ C00333 BC00333 VJ=30.00
MOVL C00334 BC00334 V=500.0
MOVL C00335 BC00335 V=500.0
'------------------------
'W62.20
'------------------------
SFTON P0358
MOVL C00336 BC00336 V=166.7 PL=0
ARCON
MOVL C00337 BC00337 V=10.0
ARCOF
MOVL C00338 BC00338 V=250.0 PL=0
SFTOF
'PRZEJAZD
MOVL C00339 BC00339 V=500.0
'------------------------
'W63.23
'------------------------
SFTON P0359
MOVL C00340 BC00340 V=166.7 PL=0
ARCON
MOVL C00341 BC00341 V=10.0
ARCOF
MOVL C00342 BC00342 V=250.0 PL=0
MOVL C00343 BC00343 V=500.0
'------------------------
'W29.29
'------------------------
SFTON P0360
MOVL C00344 BC00344 V=166.7 PL=0
ARCON
MOVL C00345 BC00345 V=10.0
ARCOF
MOVL C00346 BC00346 V=250.0 PL=0
SFTOF
'PRZEJAZD
MOVL C00347 BC00347 V=500.0
SFTON P0361
MOVL C00348 BC00348 V=166.7 PL=0
ARCON
MOVL C00349 BC00349 V=10.0
ARCOF
MOVL C00350 BC00350 V=250.0 PL=0
SFTOF
'------------------------
'W29.32
'------------------------
'PRZEJAZD
MOVL C00351 BC00351 V=500.0
MOVJ C00352 BC00352 VJ=10.00
MOVL C00353 BC00353 V=416.7
SFTON P0362
MOVL C00354 BC00354 V=166.7 PL=0
ARCON
MOVL C00355 BC00355 V=10.0
ARCOF
MOVL C00356 BC00356 V=250.0 PL=0
SFTOF
MOVL C00357 BC00357 V=250.0
SFTON P0380
MOVL C00358 BC00358 V=250.0
ARCON
MOVL C00359 BC00359 V=10.0
ARCOF
SFTOF
MOVL C00360 BC00360 V=250.0
MOVJ C00361 BC00361 VJ=20.00
MOVJ C00362 BC00362 VJ=30.00
MOVJ C00363 BC00363 VJ=30.00
MOVJ C00364 BC00364 VJ=15.00
MOVL C00365 BC00365 V=166.7
SFTON P0363
MOVL C00366 BC00366 V=166.7 PL=0
ARCON
MOVL C00367 BC00367 V=10.0
ARCOF
MOVL C00368 BC00368 V=250.0 PL=0
SFTOF
SFTON P0364
MOVL C00369 BC00369 V=166.7 PL=0
ARCON
MOVL C00370 BC00370 V=10.0
ARCOF
MOVL C00371 BC00371 V=250.0 PL=0
SFTOF
MOVJ C00372 BC00372 VJ=20.00
MOVJ C00373 BC00373 VJ=30.00
MOVJ C00374 BC00374 VJ=30.00
CALL JOB:MOVE_OUT_OF_TUNNEL
CALL JOB:CLEAN-R1
CALL JOB:MOVE_INTO_TUNNEL
'KONIEC SPAWANIA WEW STRONA
MOVJ C00375 BC00375 VJ=10.00
MOVJ C00376 BC00376 VJ=10.00
MOVJ C00377 BC00377 VJ=20.00
MOVJ C00378 BC00378 VJ=20.00
MOVJ C00379 BC00379 VJ=10.00
MOVJ C00380 BC00380 VJ=10.00
'------------------------
'W29.2
'------------------------
MOVL C00381 BC00381 V=500.0
'------------------------
'W63.5
'------------------------
SFTOF
MOVL C00382 BC00382 V=166.7 PL=0
REFP 3 C00383 BC00383
CALL JOB:SEARCH-R1
IMOV P0056 V=50.0 PL=0
SET P0301 P0006
SFTON P0301
REFP 3 C00384 BC00384
CALL JOB:SEARCH-R1
SET P0301 P0006
SFTON P0301
MOVL C00385 BC00385 V=166.7 PL=0
SFTOF
MOVL C00386 BC00386 V=500.0
MOVL C00387 BC00387 V=166.7 PL=0
REFP 3 C00388 BC00388
CALL JOB:SEARCH-R1
IMOV P0056 V=50.0 PL=0
SET P0302 P0006
SFTON P0302
REFP 3 C00389 BC00389
CALL JOB:SEARCH-R1
SET P0302 P0006
SFTON P0302
MOVL C00390 BC00390 V=166.7 PL=0
SFTOF
MOVL C00391 BC00391 V=500.0
MOVL C00392 BC00392 V=166.7 PL=0
REFP 3 C00393 BC00393
CALL JOB:SEARCH-R1
IMOV P0056 V=50.0 PL=0
SET P0303 P0006
SFTON P0303
REFP 3 C00394 BC00394
CALL JOB:SEARCH-R1
SET P0303 P0006
SFTON P0303
SFTOF
MOVL C00395 BC00395 V=166.7 PL=0
MOVL C00396 BC00396 V=500.0
MOVJ C00397 BC00397 VJ=30.00
MOVJ C00398 BC00398 VJ=30.00
MOVJ C00399 BC00399 VJ=20.00
MOVJ C00400 BC00400 VJ=30.00
MOVL C00401 BC00401 V=500.0
'------------------------
'W29.14
'------------------------
MOVL C00402 BC00402 V=166.7 PL=0
REFP 3 C00403 BC00403
CALL JOB:SEARCH-R1
IMOV P0056 V=23.0 PL=0
SET P0304 P0006
SFTON P0304
REFP 3 C00404 BC00404
CALL JOB:SEARCH-R1
SET P0304 P0006
SFTON P0304
MOVL C00405 BC00405 V=66.7 PL=0
SFTOF
'PRZEJAZD
MOVL C00406 BC00406 V=500.0
MOVL C00407 BC00407 V=500.0
'------------------------
'W63.17
'------------------------
MOVL C00408 BC00408 V=166.7 PL=0
REFP 3 C00409 BC00409
CALL JOB:SEARCH-R1
IMOV P0056 V=23.0 PL=0
SET P0305 P0006
SFTON P0305
REFP 3 C00410 BC00410
CALL JOB:SEARCH-R1
SET P0305 P0006
SFTON P0305
MOVL C00411 BC00411 V=166.7 PL=0
SFTOF
MOVL C00412 BC00412 V=500.0
MOVL C00413 BC00413 V=166.7
REFP 3 C00414 BC00414
CALL JOB:SEARCH-R1
IMOV P0056 V=23.0 PL=0
SET P0306 P0006
SFTON P0306
REFP 3 C00415 BC00415
CALL JOB:SEARCH-R1
SET P0306 P0006
SFTON P0306
MOVL C00416 BC00416 V=166.7 PL=0
'PRZEJAZD
MOVL C00417 BC00417 V=500.0
MOVL C00418 BC00418 V=166.7
REFP 3 C00419 BC00419
CALL JOB:SEARCH-R1
IMOV P0056 V=23.0 PL=0
SET P0307 P0006
SFTON P0307
REFP 3 C00420 BC00420
CALL JOB:SEARCH-R1
SET P0307 P0006
SFTON P0307
MOVL C00421 BC00421 V=166.7 PL=0
SFTOF
MOVJ C00422 BC00422 VJ=20.00
MOVJ C00423 BC00423 VJ=20.00
MOVJ C00424 BC00424 VJ=30.00
MOVJ C00425 BC00425 VJ=30.00
MOVL C00426 BC00426 V=500.0
'------------------------
'W63.20
'------------------------
MOVL C00427 BC00427 V=166.7 PL=0
REFP 3 C00428 BC00428
CALL JOB:SEARCH-R1
IMOV P0056 V=23.0 PL=0
SET P0308 P0006
SFTON P0308
REFP 3 C00429 BC00429
CALL JOB:SEARCH-R1
SET P0308 P0006
SFTON P0308
MOVL C00430 BC00430 V=166.7 PL=0
SFTOF
'PRZEJAZD
MOVL C00431 BC00431 V=500.0
'------------------------
'W63.23
'------------------------
MOVL C00432 BC00432 V=166.7 PL=0
REFP 3 C00433 BC00433
CALL JOB:SEARCH-R1
IMOV P0056 V=23.0 PL=0
SET P0309 P0006
SFTON P0309
REFP 3 C00434 BC00434
CALL JOB:SEARCH-R1
SET P0309 P0006
SFTON P0309
MOVL C00435 BC00435 V=250.0 PL=0
SFTOF
MOVL C00436 BC00436 V=500.0
MOVL C00437 BC00437 V=166.7 PL=0
REFP 3 C00438 BC00438
CALL JOB:SEARCH-R1
IMOV P0056 V=23.0 PL=0
SET P0310 P0006
SFTON P0310
REFP 3 C00439 BC00439
CALL JOB:SEARCH-R1
SET P0310 P0006
SFTON P0310
MOVL C00440 BC00440 V=250.0 PL=0
SFTOF
MOVL C00441 BC00441 V=500.0
MOVL C00442 BC00442 V=166.7 PL=0
REFP 3 C00443 BC00443
CALL JOB:SEARCH-R1
IMOV P0056 V=23.0 PL=0
SET P0311 P0006
SFTON P0311
REFP 3 C00444 BC00444
CALL JOB:SEARCH-R1
SET P0311 P0006
SFTON P0311
MOVL C00445 BC00445 V=250.0 PL=0
SFTOF
MOVL C00446 BC00446 V=500.0
MOVL C00447 BC00447 V=500.0
MOVL C00448 BC00448 V=333.3
'------------------------
'W29.29
'------------------------
MOVL C00449 BC00449 V=166.7 PL=0
REFP 3 C00450 BC00450
CALL JOB:SEARCH-R1
IMOV P0056 V=23.0 PL=0
SET P0312 P0006
SFTON P0312
REFP 3 C00451 BC00451
CALL JOB:SEARCH-R1
SET P0312 P0006
SFTON P0312
MOVL C00452 BC00452 V=250.0 PL=0
SFTOF
MOVL C00453 BC00453 V=250.0
MOVL C00454 BC00454 V=166.7 PL=0
REFP 3 C00455 BC00455
CALL JOB:SEARCH-R1
IMOV P0056 V=23.0 PL=0
SET P0318 P0006
SFTON P0318
REFP 3 C00456 BC00456
CALL JOB:SEARCH-R1
SET P0318 P0006
SFTON P0318
MOVL C00457 BC00457 V=250.0 PL=0
SFTOF
'PRZEJAZD
MOVL C00458 BC00458 V=333.3
'PRZEJAZD
MOVL C00459 BC00459 V=500.0
MOVL C00460 BC00460 V=500.0
MOVL C00461 BC00461 V=333.3
MOVL C00462 BC00462 V=333.3
MOVL C00463 BC00463 V=166.7 PL=0
REFP 3 C00464 BC00464
CALL JOB:SEARCH-R1
IMOV P0056 V=23.0 PL=0
SET P0313 P0006
SFTON P0313
REFP 3 C00465 BC00465
CALL JOB:SEARCH-R1
SET P0313 P0006
SFTON P0313
MOVL C00466 BC00466 V=250.0 PL=0
SFTOF
MOVL C00467 BC00467 V=333.3
MOVL C00468 BC00468 V=166.7 PL=0
REFP 3 C00469 BC00469
CALL JOB:SEARCH-R1
IMOV P0056 V=23.0 PL=0
SET P0314 P0006
SFTON P0314
REFP 3 C00470 BC00470
CALL JOB:SEARCH-R1
SET P0314 P0006
SFTON P0314
MOVL C00471 BC00471 V=250.0 PL=0
SFTOF
MOVJ C00472 BC00472 VJ=10.00
MOVJ C00473 BC00473 VJ=10.00
MOVJ C00474 BC00474 VJ=20.00
MOVJ C00475 BC00475 VJ=50.00
MOVJ C00476 BC00476 VJ=20.00
MOVJ C00477 BC00477 VJ=10.00
'------------------------
'W28.2
'------------------------
MOVJ C00478 BC00478 VJ=10.00
MOVJ C00479 BC00479 VJ=10.00
MOVL C00480 BC00480 V=500.0
MOVL C00481 BC00481 V=500.0
'------------------------
'W62.5
'------------------------
MOVL C00482 BC00482 V=166.7 PL=0
REFP 3 C00483 BC00483
CALL JOB:SEARCH-R1
IMOV P0056 V=23.0 PL=0
SET P0351 P0006
SFTON P0351
REFP 3 C00484 BC00484
CALL JOB:SEARCH-R1
SET P0351 P0006
SFTON P0351
MOVL C00485 BC00485 V=250.0 PL=0
SFTOF
'PRZEJAZD
MOVL C00486 BC00486 V=500.0
MOVL C00487 BC00487 V=500.0
MOVL C00488 BC00488 V=500.0
MOVL C00489 BC00489 V=166.7 PL=0
REFP 3 C00490 BC00490
CALL JOB:SEARCH-R1
IMOV P0056 V=23.0 PL=0
SET P0352 P0006
SFTON P0352
REFP 3 C00491 BC00491
CALL JOB:SEARCH-R1
SET P0352 P0006
SFTON P0352
MOVL C00492 BC00492 V=250.0 PL=0
SFTOF
MOVL C00493 BC00493 V=500.0
'------------------------
'W29.8
'------------------------
MOVL C00494 BC00494 V=166.7 PL=0
REFP 3 C00495 BC00495
CALL JOB:SEARCH-R1
IMOV P0056 V=23.0 PL=0
SET P0353 P0006
SFTON P0353
REFP 3 C00496 BC00496
CALL JOB:SEARCH-R1
SET P0353 P0006
SFTON P0353
MOVL C00497 BC00497 V=250.0 PL=0
SFTOF
MOVL C00498 BC00498 V=500.0
'PRZEJAZD
MOVL C00499 BC00499 V=500.0
MOVJ C00500 BC00500 VJ=20.00
MOVJ C00501 BC00501 VJ=20.00
MOVL C00502 BC00502 V=500.0
MOVL C00503 BC00503 V=500.0
MOVL C00504 BC00504 V=500.0
'------------------------
'W29.11
'------------------------
MOVL C00505 BC00505 V=166.7 PL=0
REFP 3 C00506 BC00506
CALL JOB:SEARCH-R1
IMOV P0056 V=23.0 PL=0
SET P0354 P0006
SFTON P0354
REFP 3 C00507 BC00507
CALL JOB:SEARCH-R1
SET P0354 P0006
SFTON P0354
MOVL C00508 BC00508 V=250.0 PL=0
SFTOF
'PRZEJAZD
MOVL C00509 BC00509 V=500.0
'------------------------
'W29.14
'------------------------
MOVL C00510 BC00510 V=166.7 PL=0
REFP 3 C00511 BC00511
CALL JOB:SEARCH-R1
IMOV P0056 V=23.0 PL=0
SET P0355 P0006
SFTON P0355
REFP 3 C00512 BC00512
CALL JOB:SEARCH-R1
SET P0355 P0006
SFTON P0355
MOVL C00513 BC00513 V=250.0 PL=0
SFTOF
'PRZEJAZD
MOVL C00514 BC00514 V=500.0
'------------------------
'W63.17
'------------------------
MOVL C00515 BC00515 V=166.7 PL=0
REFP 3 C00516 BC00516
CALL JOB:SEARCH-R1
IMOV P0056 V=23.0 PL=0
SET P0356 P0006
SFTON P0356
REFP 3 C00517 BC00517
CALL JOB:SEARCH-R1
SET P0356 P0006
SFTON P0356
MOVL C00518 BC00518 V=250.0 PL=0
SFTOF
MOVL C00519 BC00519 V=500.0
MOVL C00520 BC00520 V=166.7 PL=0
REFP 3 C00521 BC00521
CALL JOB:SEARCH-R1
IMOV P0056 V=23.0 PL=0
SET P0357 P0006
SFTON P0357
REFP 3 C00522 BC00522
CALL JOB:SEARCH-R1
SET P0357 P0006
SFTON P0357
MOVL C00523 BC00523 V=250.0 PL=0
SFTOF
'PRZEJAZD
MOVL C00524 BC00524 V=500.0
MOVJ C00525 BC00525 VJ=30.00
MOVJ C00526 BC00526 VJ=30.00
MOVL C00527 BC00527 V=500.0
MOVL C00528 BC00528 V=500.0
'------------------------
'W62.20
'------------------------
MOVL C00529 BC00529 V=166.7 PL=0
REFP 3 C00530 BC00530
CALL JOB:SEARCH-R1
IMOV P0056 V=23.0 PL=0
SET P0358 P0006
SFTON P0358
REFP 3 C00531 BC00531
CALL JOB:SEARCH-R1
SET P0358 P0006
SFTON P0358
MOVL C00532 BC00532 V=250.0 PL=0
SFTOF
'PRZEJAZD
MOVL C00533 BC00533 V=500.0
'------------------------
'W63.23
'------------------------
MOVL C00534 BC00534 V=166.7 PL=0
REFP 3 C00535 BC00535
CALL JOB:SEARCH-R1
IMOV P0056 V=23.0 PL=0
SET P0359 P0006
SFTON P0359
REFP 3 C00536 BC00536
CALL JOB:SEARCH-R1
SET P0359 P0006
SFTON P0359
MOVL C00537 BC00537 V=250.0 PL=0
MOVL C00538 BC00538 V=500.0
'------------------------
'W29.29
'------------------------
MOVL C00539 BC00539 V=166.7 PL=0
REFP 3 C00540 BC00540
CALL JOB:SEARCH-R1
IMOV P0056 V=23.0 PL=0
SET P0360 P0006
SFTON P0360
REFP 3 C00541 BC00541
CALL JOB:SEARCH-R1
SET P0360 P0006
SFTON P0360
MOVL C00542 BC00542 V=250.0 PL=0
SFTOF
'PRZEJAZD
MOVL C00543 BC00543 V=500.0
MOVL C00544 BC00544 V=166.7 PL=0
REFP 3 C00545 BC00545
CALL JOB:SEARCH-R1
IMOV P0056 V=23.0 PL=0
SET P0361 P0006
SFTON P0361
REFP 3 C00546 BC00546
CALL JOB:SEARCH-R1
SET P0361 P0006
SFTON P0361
MOVL C00547 BC00547 V=250.0 PL=0
SFTOF
'------------------------
'W29.32
'------------------------
'PRZEJAZD
MOVL C00548 BC00548 V=500.0
MOVJ C00549 BC00549 VJ=10.00
MOVL C00550 BC00550 V=416.7
MOVL C00551 BC00551 V=166.7 PL=0
REFP 3 C00552 BC00552
CALL JOB:SEARCH-R1
IMOV P0056 V=23.0 PL=0
SET P0362 P0006
SFTON P0362
REFP 3 C00553 BC00553
CALL JOB:SEARCH-R1
SET P0362 P0006
SFTON P0362
MOVL C00554 BC00554 V=250.0 PL=0
SFTOF
MOVL C00555 BC00555 V=250.0
MOVL C00556 BC00556 V=166.7 PL=0
REFP 3 C00557 BC00557
CALL JOB:SEARCH-R1
IMOV P0056 V=23.0 PL=0
SET P0380 P0006
SFTON P0380
REFP 3 C00558 BC00558
CALL JOB:SEARCH-R1
SET P0380 P0006
SFTON P0380
MOVL C00559 BC00559 V=250.0 PL=0
SFTOF
MOVJ C00560 BC00560 VJ=20.00
MOVJ C00561 BC00561 VJ=30.00
MOVJ C00562 BC00562 VJ=15.00
MOVJ C00563 BC00563 VJ=15.00
MOVL C00564 BC00564 V=166.7
MOVL C00565 BC00565 V=166.7 PL=0
REFP 3 C00566 BC00566
CALL JOB:SEARCH-R1
IMOV P0056 V=23.0 PL=0
SET P0363 P0006
SFTON P0363
REFP 3 C00567 BC00567
CALL JOB:SEARCH-R1
SET P0363 P0006
SFTON P0363
MOVL C00568 BC00568 V=250.0 PL=0
SFTOF
MOVL C00569 BC00569 V=166.7 PL=0
REFP 3 C00570 BC00570
CALL JOB:SEARCH-R1
IMOV P0056 V=23.0 PL=0
SET P0364 P0006
SFTON P0364
REFP 3 C00571 BC00571
CALL JOB:SEARCH-R1
SET P0364 P0006
SFTON P0364
MOVL C00572 BC00572 V=250.0 PL=0
SFTOF
MOVJ C00573 BC00573 VJ=20.00
MOVJ C00574 BC00574 VJ=30.00
MOVJ C00575 BC00575 VJ=30.00
'KONIEC SEARCH ZEW STRONA
MOVJ C00576 BC00576 VJ=30.00
MOVJ C00577 BC00577 VJ=20.00
MOVJ C00578 BC00578 VJ=10.00
MOVJ C00579 BC00579 VJ=20.00
MOVJ C00580 BC00580 VJ=20.00
'------------------------
'W29.2
'------------------------
MOVL C00581 BC00581 V=500.0
'------------------------
'W63.5
MACRO1 MJ#(0) ARGF9
'------------------------
SFTOF
SFTON P0301
MOVL C00582 BC00582 V=166.7 PL=0
ARCON
MOVL C00583 BC00583 V=8.3
ARCOF
SFTOF
MOVL C00584 BC00584 V=500.0
MACRO1 MJ#(0) ARGF24
SFTON P0302
MOVL C00585 BC00585 V=166.7 PL=0
ARCON
MOVL C00586 BC00586 V=8.3
ARCOF
MOVL C00587 BC00587 V=166.7 PL=0
SFTOF
MOVL C00588 BC00588 V=500.0
SFTON P0303
MOVL C00589 BC00589 V=166.7 PL=0
ARCON
MOVL C00590 BC00590 V=8.3
ARCOF
SFTOF
MOVL C00591 BC00591 V=166.7 PL=0
MOVL C00592 BC00592 V=500.0
MOVJ C00593 BC00593 VJ=30.00
MOVJ C00594 BC00594 VJ=20.00
MOVJ C00595 BC00595 VJ=30.00
MOVJ C00596 BC00596 VJ=30.00
MOVL C00597 BC00597 V=500.0
'------------------------
'W29.14
'------------------------
SFTON P0304
MOVL C00598 BC00598 V=166.7 PL=0
ARCON
MOVL C00599 BC00599 V=8.3
ARCOF
MOVL C00600 BC00600 V=166.7 PL=0
SFTOF
'PRZEJAZD
MOVL C00601 BC00601 V=500.0
MOVL C00602 BC00602 V=500.0
'------------------------
'W63.17
'------------------------
SFTON P0305
MOVL C00603 BC00603 V=166.7 PL=0
ARCON
MOVL C00604 BC00604 V=8.3
ARCOF
MOVL C00605 BC00605 V=166.7 PL=0
SFTOF
MOVL C00606 BC00606 V=500.0
SFTON P0306
MOVL C00607 BC00607 V=166.7
ARCON
MOVL C00608 BC00608 V=8.3
ARCOF
MOVL C00609 BC00609 V=166.7 PL=0
SFTOF
'PRZEJAZD
MOVL C00610 BC00610 V=500.0
SFTON P0307
MOVL C00611 BC00611 V=166.7
ARCON
MOVL C00612 BC00612 V=8.3
ARCOF
MOVL C00613 BC00613 V=166.7 PL=0
SFTOF
MOVJ C00614 BC00614 VJ=20.00
MOVJ C00615 BC00615 VJ=20.00
MOVJ C00616 BC00616 VJ=30.00
MOVJ C00617 BC00617 VJ=30.00
MOVL C00618 BC00618 V=500.0
'------------------------
'W63.20
'------------------------
SFTON P0308
MOVL C00619 BC00619 V=166.7 PL=0
ARCON
MOVL C00620 BC00620 V=8.3
ARCOF
MOVL C00621 BC00621 V=166.7 PL=0
SFTOF
'PRZEJAZD
MOVL C00622 BC00622 V=500.0
'------------------------
'W63.23
'------------------------
SFTON P0309
MOVL C00623 BC00623 V=166.7 PL=0
ARCON
MOVL C00624 BC00624 V=8.3
ARCOF
MOVL C00625 BC00625 V=250.0 PL=0
SFTOF
MOVL C00626 BC00626 V=500.0
SFTON P0310
MOVL C00627 BC00627 V=166.7 PL=0
ARCON
MOVL C00628 BC00628 V=8.3
ARCOF
MOVL C00629 BC00629 V=250.0 PL=0
SFTOF
MOVL C00630 BC00630 V=500.0
SFTON P0311
MOVL C00631 BC00631 V=166.7 PL=0
ARCON
MOVL C00632 BC00632 V=8.3
ARCOF
MOVL C00633 BC00633 V=250.0 PL=0
SFTOF
MOVL C00634 BC00634 V=500.0
MOVL C00635 BC00635 V=500.0
MOVL C00636 BC00636 V=333.3
'------------------------
'W29.29
'------------------------
SFTON P0312
MOVL C00637 BC00637 V=166.7 PL=0
ARCON
MOVL C00638 BC00638 V=8.3
ARCOF
MOVL C00639 BC00639 V=250.0 PL=0
SFTOF
MOVL C00640 BC00640 V=250.0
SFTON P0318
MOVL C00641 BC00641 V=250.0
ARCON
MOVL C00642 BC00642 V=8.3
ARCOF
SFTOF
'PRZEJAZD
MOVL C00643 BC00643 V=333.3
'PRZEJAZD
'KONIEC SPAWANIA CZESCI WSPOLNEJ
MOVL C00644 BC00644 V=500.0
MOVL C00645 BC00645 V=500.0
MOVL C00646 BC00646 V=500.0
MOVL C00647 BC00647 V=333.3
MOVL C00648 BC00648 V=333.3
SFTON P0313
MOVL C00649 BC00649 V=166.7 PL=0
ARCON
MOVL C00650 BC00650 V=8.3
ARCOF
MOVL C00651 BC00651 V=250.0 PL=0
SFTOF
MOVL C00652 BC00652 V=333.3
SFTON P0314
MOVL C00653 BC00653 V=166.7 PL=0
ARCON
MOVL C00654 BC00654 V=8.3
ARCOF
MOVL C00655 BC00655 V=250.0 PL=0
SFTOF
MOVJ C00656 BC00656 VJ=10.00
MOVJ C00657 BC00657 VJ=10.00
MOVJ C00658 BC00658 VJ=30.00
MOVJ C00659 BC00659 VJ=20.00
MOVJ C00660 BC00660 VJ=50.00
MOVJ C00661 BC00661 VJ=20.00
MOVJ C00662 BC00662 VJ=10.00
MOVJ C00663 BC00663 VJ=20.00
MOVJ C00664 BC00664 VJ=20.00
'------------------------
'W28.2
'------------------------
MOVJ C00665 BC00665 VJ=10.00
MOVJ C00666 BC00666 VJ=10.00
MOVL C00667 BC00667 V=500.0
MOVL C00668 BC00668 V=500.0
'------------------------
'W62.5
'------------------------
SFTON P0351
MOVL C00669 BC00669 V=166.7 PL=0
ARCON
MOVL C00670 BC00670 V=8.3
ARCOF
MOVL C00671 BC00671 V=250.0 PL=0
SFTOF
'PRZEJAZD
MOVL C00672 BC00672 V=500.0
MOVL C00673 BC00673 V=500.0
MOVL C00674 BC00674 V=500.0
SFTON P0352
MOVL C00675 BC00675 V=166.7 PL=0
ARCON
MOVL C00676 BC00676 V=8.3
ARCOF
MOVL C00677 BC00677 V=250.0 PL=0
SFTOF
MOVL C00678 BC00678 V=500.0
'------------------------
'W29.8
'------------------------
SFTON P0353
MOVL C00679 BC00679 V=166.7 PL=0
ARCON
MOVL C00680 BC00680 V=8.3
ARCOF
MOVL C00681 BC00681 V=250.0 PL=0
SFTOF
MOVL C00682 BC00682 V=500.0
'PRZEJAZD
MOVL C00683 BC00683 V=500.0
MOVJ C00684 BC00684 VJ=20.00
MOVL C00685 BC00685 V=500.0
MOVL C00686 BC00686 V=500.0
MOVL C00687 BC00687 V=500.0
'------------------------
'W29.11
'------------------------
SFTON P0354
MOVL C00688 BC00688 V=166.7 PL=0
ARCON
MOVL C00689 BC00689 V=8.3
ARCOF
MOVL C00690 BC00690 V=250.0 PL=0
SFTOF
'PRZEJAZD
MOVL C00691 BC00691 V=500.0
'------------------------
'W29.14
'------------------------
SFTON P0355
MOVL C00692 BC00692 V=166.7 PL=0
ARCON
MOVL C00693 BC00693 V=8.3
ARCOF
MOVL C00694 BC00694 V=250.0 PL=0
SFTOF
'PRZEJAZD
MOVL C00695 BC00695 V=500.0
'------------------------
'W63.17
'------------------------
SFTON P0356
MOVL C00696 BC00696 V=166.7 PL=0
ARCON
MOVL C00697 BC00697 V=8.3
ARCOF
MOVL C00698 BC00698 V=250.0 PL=0
SFTOF
MOVL C00699 BC00699 V=500.0
SFTON P0357
MOVL C00700 BC00700 V=166.7 PL=0
ARCON
MOVL C00701 BC00701 V=8.3
ARCOF
MOVL C00702 BC00702 V=250.0 PL=0
SFTOF
'PRZEJAZD
MOVL C00703 BC00703 V=500.0
MOVJ C00704 BC00704 VJ=30.00
MOVJ C00705 BC00705 VJ=30.00
MOVJ C00706 BC00706 VJ=30.00
MOVL C00707 BC00707 V=500.0
MOVL C00708 BC00708 V=500.0
'------------------------
'W62.20
'------------------------
SFTON P0358
MOVL C00709 BC00709 V=166.7 PL=0
ARCON
MOVL C00710 BC00710 V=8.3
ARCOF
MOVL C00711 BC00711 V=250.0 PL=0
SFTOF
'PRZEJAZD
MOVL C00712 BC00712 V=500.0
'------------------------
'W63.23
'------------------------
SFTON P0359
MOVL C00713 BC00713 V=166.7 PL=0
ARCON
MOVL C00714 BC00714 V=8.3
ARCOF
MOVL C00715 BC00715 V=250.0 PL=0
MOVL C00716 BC00716 V=500.0
'------------------------
'W29.29
'------------------------
SFTON P0360
MOVL C00717 BC00717 V=166.7 PL=0
ARCON
MOVL C00718 BC00718 V=8.3
ARCOF
MOVL C00719 BC00719 V=250.0 PL=0
SFTOF
'PRZEJAZD
MOVL C00720 BC00720 V=500.0
SFTON P0361
MOVL C00721 BC00721 V=166.7 PL=0
ARCON
MOVL C00722 BC00722 V=8.3
ARCOF
MOVL C00723 BC00723 V=250.0 PL=0
SFTOF
'------------------------
'W29.32
'------------------------
'PRZEJAZD
MOVL C00724 BC00724 V=500.0
MOVJ C00725 BC00725 VJ=10.00
MOVL C00726 BC00726 V=416.7
SFTON P0362
MOVL C00727 BC00727 V=166.7 PL=0
ARCON
MOVL C00728 BC00728 V=8.3
ARCOF
MOVL C00729 BC00729 V=250.0 PL=0
SFTOF
MOVL C00730 BC00730 V=250.0
SFTON P0380
MOVL C00731 BC00731 V=166.7
ARCON
MOVL C00732 BC00732 V=8.3
ARCOF
SFTOF
MOVL C00733 BC00733 V=250.0
MOVJ C00734 BC00734 VJ=20.00
MOVJ C00735 BC00735 VJ=30.00
MOVJ C00736 BC00736 VJ=15.00
MOVJ C00737 BC00737 VJ=15.00
MOVL C00738 BC00738 V=166.7
SFTON P0363
MOVL C00739 BC00739 V=166.7 PL=0
ARCON
MOVL C00740 BC00740 V=8.3
ARCOF
MOVL C00741 BC00741 V=250.0 PL=0
SFTOF
SFTON P0364
MOVL C00742 BC00742 V=166.7 PL=0
ARCON
MOVL C00743 BC00743 V=8.3
ARCOF
MOVL C00744 BC00744 V=250.0 PL=0
SFTOF
MOVJ C00745 BC00745 VJ=20.00
MOVJ C00746 BC00746 VJ=30.00
MOVJ C00747 BC00747 VJ=30.00
CALL JOB:MOVE_OUT_OF_TUNNEL
END
